KUKA KRL program: MyProgram_294().src

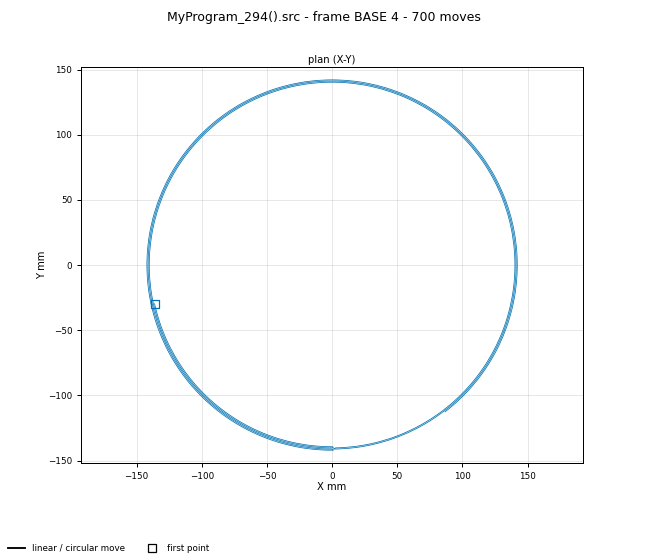
[picture p0: tool path of MyProgram_294().src in frame BASE 4, 700 of 700 moves have a stored position in this frame; points joined in program order, loops and branches not executed]
&ACCESS RVP
&REL 1
&PARAM TEMPLATE = C:\KRC\Roboter\Template\vorgabe
&PARAM EDITMASK = *
DEF MyProgram_294()
; ---- Setting reference (Base) ----
$BASE = BASE_DATA[4]

; --------------------------
; ---- Setting tool (TCP) ----
$TOOL = TOOL_DATA[3]
; --------------------------

$VEL.CP = VEL_APROX_PRINT
Startdeposition()
$VEL.CP = VEL_PRINT
LIN {X -136.1886,Y -29.6785,Z 177,A -164.7897,B 6.5614,C 0.2921,E1 6.4117,E2 257.0139} C_DIS
LIN {X -135.5022,Y -32.6682,Z 177,A -163.4829,B 6.5613,C 0.295,E1 6.4125,E2 255.702} C_DIS
LIN {X -134.5919,Y -36.238,Z 177,A -161.9756,B 6.5611,C 0.2993,E1 6.4136,E2 254.1966} C_DIS
LIN {X -133.5688,Y -39.8487,Z 177,A -160.401,B 6.5609,C 0.3031,E1 6.4148,E2 252.619} C_DIS
LIN {X -132.4479,Y -43.4282,Z 177,A -158.721,B 6.5608,C 0.3057,E1 6.4163,E2 250.9221} C_DIS
LIN {X -130.5858,Y -48.7382,Z 177,A -156.3622,B 6.5605,C 0.3113,E1 6.4185,E2 248.5587} C_DIS
LIN {X -129.1386,Y -52.4536,Z 177,A -154.7567,B 6.5603,C 0.316,E1 6.4201,E2 246.9586} C_DIS
LIN {X -127.4559,Y -56.4207,Z 177,A -152.7896,B 6.5602,C 0.3183,E1 6.4224,E2 244.9671} C_DIS
LIN {X -125.5768,Y -60.4868,Z 177,A -151.0792,B 6.5599,C 0.3246,E1 6.4244,E2 243.2747} C_DIS
LIN {X -123.9871,Y -63.6824,Z 177,A -149.5853,B 6.5597,C 0.3279,E1 6.4263,E2 241.7781} C_DIS
LIN {X -120.2753,Y -70.4446,Z 177,A -146.6108,B 6.5592,C 0.3381,E1 6.4303,E2 238.8308} C_DIS
LIN {X -117.7123,Y -74.649,Z 177,A -144.0898,B 6.5592,C 0.3369,E1 6.4341,E2 236.2462} C_DIS
LIN {X -114.5903,Y -79.3582,Z 177,A -141.8024,B 6.559,C 0.3427,E1 6.4376,E2 233.9644} C_DIS
LIN {X -111.921,Y -83.0801,Z 177,A -139.9675,B 6.5587,C 0.3476,E1 6.4406,E2 232.1365} C_DIS
LIN {X -109.4462,Y -86.3143,Z 177,A -138.2223,B 6.5586,C 0.3504,E1 6.4436,E2 230.3825} C_DIS
LIN {X -106.5575,Y -89.8563,Z 177,A -136.3073,B 6.5584,C 0.3539,E1 6.4471,E2 228.4635} C_DIS
LIN {X -103.5566,Y -93.2993,Z 177,A -134.3994,B 6.5582,C 0.3575,E1 6.4506,E2 226.5522} C_DIS
LIN {X -100.555,Y -96.5264,Z 177,A -132.5532,B 6.558,C 0.3607,E1 6.4541,E2 224.7019} C_DIS
LIN {X -97.3293,Y -99.7782,Z 177,A -130.6364,B 6.5578,C 0.3639,E1 6.458,E2 222.7812} C_DIS
LIN {X -93.9858,Y -102.9341,Z 177,A -128.6876,B 6.5577,C 0.3667,E1 6.462,E2 220.8251} C_DIS
LIN {X -90.5246,Y -105.9904,Z 177,A -126.7715,B 6.5575,C 0.3698,E1 6.466,E2 218.9069} C_DIS
LIN {X -86.9356,Y -108.9531,Z 177,A -124.8461,B 6.5573,C 0.373,E1 6.4702,E2 216.9803} C_DIS
LIN {X -83.3113,Y -111.7488,Z 177,A -122.5359,B 6.5575,C 0.3704,E1 6.4755,E2 214.6138} C_DIS
LIN {X -79.6539,Y -114.3842,Z 177,A -121.0582,B 6.557,C 0.3783,E1 6.4787,E2 213.1858} C_DIS
LIN {X -76.0946,Y -116.7827,Z 177,A -119.334,B 6.5568,C 0.3814,E1 6.4827,E2 211.4669} C_DIS
LIN {X -73.4203,Y -118.4824,Z 177,A -117.9768,B 6.5568,C 0.3825,E1 6.486,E2 210.1027} C_DIS
LIN {X -69.5459,Y -120.7975,Z 177,A -116.113,B 6.5566,C 0.3849,E1 6.4905,E2 208.2377} C_DIS
LIN {X -65.5857,Y -122.9929,Z 177,A -114.0349,B 6.5566,C 0.3843,E1 6.4956,E2 206.131} C_DIS
LIN {X -60.1602,Y -125.7329,Z 177,A -112.0219,B 6.5561,C 0.3939,E1 6.5005,E2 204.1818} C_DIS
LIN {X -56.9114,Y -127.2364,Z 177,A -110.2509,B 6.5562,C 0.3914,E1 6.5051,E2 202.3712} C_DIS
LIN {X -53.2044,Y -128.8317,Z 177,A -108.6402,B 6.5562,C 0.3937,E1 6.5093,E2 200.7667} C_DIS
LIN {X -49.6793,Y -130.2332,Z 177,A -106.9373,B 6.5562,C 0.3932,E1 6.5137,E2 199.0448} C_DIS
LIN {X -46.3018,Y -131.4711,Z 177,A -105.6473,B 6.5559,C 0.3971,E1 6.5171,E2 197.7795} C_DIS
LIN {X -43.7304,Y -132.3472,Z 177,A -104.4709,B 6.5559,C 0.3971,E1 6.5202,E2 196.5949} C_DIS
LIN {X -40.4619,Y -133.3829,Z 177,A -103.0141,B 6.5559,C 0.3975,E1 6.5241,E2 195.1316} C_DIS
LIN {X -34.6228,Y -135.0164,Z 177,A -100.724,B 6.5556,C 0.402,E1 6.5302,E2 192.8676} C_DIS
LIN {X -30.5072,Y -136.0062,Z 177,A -98.6594,B 6.5558,C 0.3982,E1 6.5359,E2 190.7597} C_DIS
LIN {X -26.4921,Y -136.8443,Z 177,A -96.9236,B 6.5558,C 0.3982,E1 6.5407,E2 189.0168} C_DIS
LIN {X -21.8811,Y -137.6576,Z 177,A -95.2757,B 6.5555,C 0.403,E1 6.5451,E2 187.405} C_DIS
LIN {X -19.1338,Y -138.0665,Z 177,A -93.9305,B 6.5557,C 0.4003,E1 6.5489,E2 186.0325} C_DIS
LIN {X -15.0645,Y -138.5684,Z 177,A -92.3262,B 6.5557,C 0.4019,E1 6.5534,E2 184.4383} C_DIS
LIN {X -11.5684,Y -138.904,Z 177,A -90.8501,B 6.5557,C 0.4016,E1 6.5575,E2 182.9572} C_DIS
LIN {X -7.1704,Y -139.2004,Z 177,A -89.0559,B 6.5557,C 0.402,E1 6.5625,E2 181.1646} C_DIS
LIN {X -3.2385,Y -139.3487,Z 177,A -87.4999,B 6.5556,C 0.4028,E1 6.5668,E2 179.6161} C_DIS
LIN {X 0.4018,Y -139.3849,Z 177,A -85.9175,B 6.5556,C 0.4014,E1 6.5713,E2 178.0216} C_DIS
LIN {X 0.4018,Y -139.3849,Z 177,A -85.9175,B 6.5556,C 0.4014,E1 6.5713,E2 178.0216} C_DIS
Enddeposition()
LIN {X 1.0085,Y -140.2847,Z 177,A -86.2982,B 6.5725,C 0.4147,E1 6.5876,E2 178.5133} C_DIS
Startdeposition()
$VEL.CP = VEL_PRINT
LIN {X -2.8125,Y -140.2623,Z 177,A -87.858,B 6.5725,C 0.4149,E1 6.5832,E2 180.0737} C_DIS
LIN {X -6.743,Y -140.1278,Z 177,A -89.5284,B 6.5725,C 0.4159,E1 6.5785,E2 181.7533} C_DIS
LIN {X -10.175,Y -139.9201,Z 177,A -90.9101,B 6.5725,C 0.4154,E1 6.5747,E2 183.1326} C_DIS
LIN {X -14.267,Y -139.5642,Z 177,A -92.617,B 6.5725,C 0.4156,E1 6.5699,E2 184.8441} C_DIS
LIN {X -18.2788,Y -139.0936,Z 177,A -94.2448,B 6.5725,C 0.4149,E1 6.5654,E2 186.4696} C_DIS
LIN {X -22.4184,Y -138.4883,Z 177,A -96.1778,B 6.5723,C 0.4176,E1 6.56,E2 188.4327} C_DIS
LIN {X -27.1842,Y -137.6328,Z 177,A -97.9321,B 6.5726,C 0.4136,E1 6.5553,E2 190.1582} C_DIS
LIN {X -29.7523,Y -137.0983,Z 177,A -99.4764,B 6.5722,C 0.4199,E1 6.5509,E2 191.7649} C_DIS
LIN {X -34.063,Y -136.092,Z 177,A -101.4743,B 6.5721,C 0.4215,E1 6.5454,E2 193.788} C_DIS
LIN {X -39.2291,Y -134.693,Z 177,A -103.0526,B 6.5727,C 0.4114,E1 6.5414,E2 195.2874} C_DIS
LIN {X -42.7662,Y -133.6119,Z 177,A -104.4674,B 6.5729,C 0.409,E1 6.5376,E2 196.6899} C_DIS
LIN {X -45.7296,Y -132.627,Z 177,A -105.8806,B 6.5729,C 0.4099,E1 6.5338,E2 198.1214} C_DIS
LIN {X -50.0559,Y -131.0578,Z 177,A -107.8843,B 6.5729,C 0.4099,E1 6.5285,E2 200.1417} C_DIS
LIN {X -53.8578,Y -129.5394,Z 177,A -109.371,B 6.5731,C 0.4057,E1 6.5248,E2 201.6042} C_DIS
LIN {X -57.9887,Y -127.7457,Z 177,A -111.3634,B 6.5731,C 0.4059,E1 6.5196,E2 203.617} C_DIS
LIN {X -61.8692,Y -125.9098,Z 177,A -113.4842,B 6.5729,C 0.4089,E1 6.5142,E2 205.7859} C_DIS
LIN {X -65.798,Y -123.9035,Z 177,A -114.8633,B 6.5734,C 0.401,E1 6.5109,E2 207.1099} C_DIS
LIN {X -69.5973,Y -121.8106,Z 177,A -116.6692,B 6.5734,C 0.3991,E1 6.5065,E2 208.9203} C_DIS
LIN {X -73.3729,Y -119.5744,Z 177,A -118.3934,B 6.5737,C 0.3958,E1 6.5024,E2 210.6356} C_DIS
LIN {X -76.9211,Y -117.3236,Z 177,A -120.2857,B 6.5737,C 0.3956,E1 6.4979,E2 212.5509} C_DIS
LIN {X -79.8082,Y -115.3794,Z 177,A -122.1332,B 6.5735,C 0.3991,E1 6.4935,E2 214.4538} C_DIS
LIN {X -83.5517,Y -112.6978,Z 177,A -123.6266,B 6.574,C 0.391,E1 6.4903,E2 215.8966} C_DIS
LIN {X -87.2512,Y -109.8583,Z 177,A -125.5322,B 6.5742,C 0.3878,E1 6.4861,E2 217.802} C_DIS
LIN {X -90.6845,Y -107.042,Z 177,A -127.391,B 6.5743,C 0.3852,E1 6.4821,E2 219.6664} C_DIS
LIN {X -94.1044,Y -104.0482,Z 177,A -129.264,B 6.5745,C 0.382,E1 6.4782,E2 221.5413} C_DIS
LIN {X -97.3565,Y -101.012,Z 177,A -131.1315,B 6.5747,C 0.3792,E1 6.4744,E2 223.4149} C_DIS
LIN {X -100.5963,Y -97.7858,Z 177,A -132.9829,B 6.5749,C 0.3753,E1 6.4707,E2 225.2637} C_DIS
LIN {X -103.5666,Y -94.6348,Z 177,A -134.8172,B 6.575,C 0.3726,E1 6.4672,E2 227.1061} C_DIS
LIN {X -106.631,Y -91.1679,Z 177,A -136.7244,B 6.5752,C 0.3688,E1 6.4637,E2 229.0149} C_DIS
LIN {X -109.532,Y -87.6612,Z 177,A -138.6414,B 6.5754,C 0.3655,E1 6.4603,E2 230.9388} C_DIS
LIN {X -112.3124,Y -84.0694,Z 177,A -140.5108,B 6.5756,C 0.3616,E1 6.4572,E2 232.8094} C_DIS
LIN {X -114.9528,Y -80.4213,Z 177,A -142.3794,B 6.5759,C 0.3578,E1 6.4541,E2 234.681} C_DIS
LIN {X -117.1431,Y -77.1953,Z 177,A -144.0543,B 6.5759,C 0.3551,E1 6.4515,E2 236.3659} C_DIS
LIN {X -119.6121,Y -73.3114,Z 177,A -145.7907,B 6.5763,C 0.3488,E1 6.449,E2 238.0829} C_DIS
LIN {X -123.8959,Y -65.8125,Z 177,A -149.4945,B 6.5767,C 0.3424,E1 6.4439,E2 241.808} C_DIS
LIN {X -125.6351,Y -62.4261,Z 177,A -151.0129,B 6.5769,C 0.338,E1 6.442,E2 243.3209} C_DIS
LIN {X -127.1911,Y -59.1911,Z 177,A -152.4543,B 6.5771,C 0.334,E1 6.4403,E2 244.7583} C_DIS
LIN {X -128.6405,Y -55.9712,Z 177,A -153.9384,B 6.5773,C 0.3307,E1 6.4386,E2 246.2469} C_DIS
LIN {X -130.8187,Y -50.671,Z 177,A -156.8492,B 6.5773,C 0.3313,E1 6.4355,E2 249.2297} C_DIS
LIN {X -132.3843,Y -46.4297,Z 177,A -158.2114,B 6.5778,C 0.3207,E1 6.4343,E2 250.5287} C_DIS
LIN {X -133.6222,Y -42.7338,Z 177,A -159.731,B 6.578,C 0.3155,E1 6.433,E2 252.0379} C_DIS
LIN {X -134.5625,Y -39.6748,Z 177,A -161.1596,B 6.5781,C 0.3134,E1 6.4318,E2 253.4813} C_DIS
LIN {X -135.53,Y -36.2316,Z 177,A -162.6621,B 6.5783,C 0.3099,E1 6.4307,E2 254.9882} C_DIS
LIN {X -136.2845,Y -33.2837,Z 177,A -163.8535,B 6.5785,C 0.3059,E1 6.4299,E2 256.1722} C_DIS
LIN {X -137.0587,Y -29.9357,Z 177,A -165.4547,B 6.5785,C 0.3043,E1 6.4289,E2 257.7977} C_DIS
LIN {X -137.8097,Y -26.2605,Z 177,A -167.033,B 6.5787,C 0.3005,E1 6.428,E2 259.3809} C_DIS
LIN {X -138.6022,Y -21.6941,Z 177,A -168.7747,B 6.579,C 0.2935,E1 6.4272,E2 261.1019} C_DIS
LIN {X -139.1207,Y -18.0721,Z 177,A -170.3783,B 6.5792,C 0.2905,E1 6.4266,E2 262.7184} C_DIS
LIN {X -139.8977,Y -10.4823,Z 177,A -173.7243,B 6.5794,C 0.2843,E1 6.4257,E2 266.0915} C_DIS
LIN {X -140.2454,Y -3.5444,Z 177,A -177.3186,B 6.5794,C 0.2848,E1 6.4254,E2 269.7794} C_DIS
LIN {X -140.2664,Y 2.5688,Z 177,A -178.7161,B 6.5802,C 0.2651,E1 6.4254,E2 271.0353} C_DIS
LIN {X -139.9234,Y 10.1302,Z 177,A 178.0725,B 6.5805,C 0.2577,E1 6.4258,E2 274.2598} C_DIS
LIN {X -139.2431,Y 17.1104,Z 177,A 174.739,B 6.5806,C 0.255,E1 6.4268,E2 277.6509} C_DIS
LIN {X -138.3679,Y 23.1403,Z 177,A 171.8862,B 6.5807,C 0.252,E1 6.428,E2 280.5476} C_DIS
LIN {X -137.6263,Y 27.216,Z 177,A 170.4757,B 6.581,C 0.2441,E1 6.4287,E2 281.9211} C_DIS
LIN {X -136.9099,Y 30.6138,Z 177,A 169.0511,B 6.5812,C 0.2402,E1 6.4296,E2 283.3452} C_DIS
LIN {X -136.0591,Y 34.1924,Z 177,A 167.6831,B 6.5814,C 0.2344,E1 6.4305,E2 284.6948} C_DIS
LIN {X -135.1271,Y 37.7063,Z 177,A 166.2172,B 6.5815,C 0.2301,E1 6.4315,E2 286.157} C_DIS
LIN {X -134.2419,Y 40.7467,Z 177,A 164.7417,B 6.5815,C 0.2286,E1 6.4327,E2 287.6544} C_DIS
LIN {X -133.1815,Y 44.0888,Z 177,A 163.3748,B 6.5817,C 0.2239,E1 6.4339,E2 289.0117} C_DIS
LIN {X -131.9466,Y 47.6568,Z 177,A 161.6628,B 6.5818,C 0.2217,E1 6.4355,E2 290.7439} C_DIS
LIN {X -130.9111,Y 50.4334,Z 177,A 160.116,B 6.5818,C 0.2224,E1 6.4371,E2 292.3319} C_DIS
LIN {X -129.5508,Y 53.8303,Z 177,A 158.8562,B 6.582,C 0.2157,E1 6.4384,E2 293.5609} C_DIS
LIN {X -128.054,Y 57.2994,Z 177,A 157.0507,B 6.582,C 0.2147,E1 6.4405,E2 295.3979} C_DIS
LIN {X -126.5856,Y 60.4743,Z 177,A 156.2293,B 6.5824,C 0.2039,E1 6.4413,E2 296.1414} C_DIS
LIN {X -123.4294,Y 66.6851,Z 177,A 152.923,B 6.5824,C 0.2021,E1 6.4456,E2 299.5036} C_DIS
LIN {X -121.1896,Y 70.6744,Z 177,A 151.0247,B 6.5826,C 0.1977,E1 6.4483,E2 301.4039} C_DIS
LIN {X -118.9135,Y 74.4401,Z 177,A 149.1789,B 6.5826,C 0.1939,E1 6.451,E2 303.2542} C_DIS
LIN {X -116.4482,Y 78.2406,Z 177,A 147.2803,B 6.5828,C 0.1901,E1 6.4539,E2 305.1572} C_DIS
LIN {X -113.8534,Y 81.9707,Z 177,A 145.3894,B 6.5829,C 0.1861,E1 6.4569,E2 307.0508} C_DIS
LIN {X -111.5269,Y 85.1079,Z 177,A 143.6904,B 6.5829,C 0.1837,E1 6.4598,E2 308.7614} C_DIS
LIN {X -108.3748,Y 89.088,Z 177,A 141.8945,B 6.5832,C 0.1757,E1 6.4629,E2 310.5205} C_DIS
LIN {X -104.715,Y 93.362,Z 177,A 138.5732,B 6.583,C 0.1831,E1 6.4693,E2 313.9674} C_DIS
LIN {X -100.3605,Y 98.0278,Z 177,A 136.9969,B 6.5835,C 0.1652,E1 6.4721,E2 315.4129} C_DIS
LIN {X -97.366,Y 101.0014,Z 177,A 134.8187,B 6.5835,C 0.1673,E1 6.4765,E2 317.6467} C_DIS
LIN {X -90.5016,Y 107.1973,Z 177,A 131.1066,B 6.5836,C 0.1594,E1 6.4842,E2 321.3474} C_DIS
LIN {X -85.6784,Y 111.0897,Z 177,A 128.1756,B 6.5836,C 0.1598,E1 6.4908,E2 324.3261} C_DIS
LIN {X -82.3284,Y 113.5942,Z 177,A 126.7409,B 6.5838,C 0.1535,E1 6.4939,E2 325.7253} C_DIS
LIN {X -78.3518,Y 116.3732,Z 177,A 124.7895,B 6.5838,C 0.15,E1 6.4984,E2 327.6714} C_DIS
LIN {X -74.5441,Y 118.8484,Z 177,A 122.9372,B 6.5839,C 0.1471,E1 6.5027,E2 329.5219} C_DIS
LIN {X -70.8056,Y 121.1126,Z 177,A 121.1103,B 6.5839,C 0.145,E1 6.5071,E2 331.3525} C_DIS
LIN {X -67.0507,Y 123.2308,Z 177,A 119.354,B 6.584,C 0.1425,E1 6.5114,E2 333.107} C_DIS
LIN {X -63.9541,Y 124.864,Z 177,A 118.0702,B 6.584,C 0.1387,E1 6.5146,E2 334.3712} C_DIS
LIN {X -59.7043,Y 126.9534,Z 177,A 115.932,B 6.584,C 0.139,E1 6.52,E2 336.5336} C_DIS
LIN {X -56.2081,Y 128.5381,Z 177,A 114.5409,B 6.5842,C 0.1349,E1 6.5235,E2 337.9015} C_DIS
LIN {X -54.0951,Y 129.4402,Z 177,A 113.0331,B 6.584,C 0.1413,E1 6.5276,E2 339.4795} C_DIS
LIN {X -49.957,Y 131.0954,Z 177,A 111.6943,B 6.5842,C 0.1331,E1 6.5309,E2 340.7572} C_DIS
LIN {X -46.3635,Y 132.4073,Z 177,A 110.118,B 6.5842,C 0.1318,E1 6.535,E2 342.3341} C_DIS
LIN {X -42.7693,Y 133.6109,Z 177,A 108.5781,B 6.5842,C 0.1303,E1 6.5391,E2 343.8719} C_DIS
LIN {X -40.1654,Y 134.4189,Z 177,A 107.3146,B 6.5842,C 0.1315,E1 6.5425,E2 345.1535} C_DIS
LIN {X -35.8988,Y 135.6187,Z 177,A 105.4528,B 6.5842,C 0.1308,E1 6.5476,E2 347.0206} C_DIS
LIN {X -31.5,Y 136.7075,Z 177,A 103.751,B 6.5843,C 0.1276,E1 6.5521,E2 348.7026} C_DIS
LIN {X -26.0009,Y 137.8594,Z 177,A 101.4275,B 6.5843,C 0.1267,E1 6.5585,E2 351.0283} C_DIS
LIN {X -19.8062,Y 138.8844,Z 177,A 98.8473,B 6.5843,C 0.1258,E1 6.5656,E2 353.6091} C_DIS
LIN {X -16.1577,Y 139.3567,Z 177,A 97.3523,B 6.5843,C 0.1252,E1 6.5698,E2 355.1024} C_DIS
LIN {X -10.6382,Y 139.8863,Z 177,A 95.0449,B 6.5843,C 0.1252,E1 6.5762,E2 357.414} C_DIS
LIN {X -6.0192,Y 140.1616,Z 177,A 93.1305,B 6.5843,C 0.1254,E1 6.5815,E2 359.3306} C_DIS
LIN {X -2.6617,Y 140.2649,Z 177,A 91.7806,B 6.5843,C 0.125,E1 6.5853,E2 360.677} C_DIS
LIN {X 1.2875,Y 140.2848,Z 177,A 90.1404,B 6.5843,C 0.1254,E1 6.5899,E2 362.32} C_DIS
LIN {X 5.4175,Y 140.1851,Z 177,A 88.5025,B 6.5843,C 0.1249,E1 6.5944,E2 363.951} C_DIS
LIN {X 9.1341,Y 139.9929,Z 177,A 86.9392,B 6.5843,C 0.1258,E1 6.5988,E2 365.5191} C_DIS
LIN {X 13.3698,Y 139.6511,Z 177,A 85.2082,B 6.5843,C 0.1262,E1 6.6036,E2 367.2489} C_DIS
LIN {X 16.9885,Y 139.2576,Z 177,A 83.1093,B 6.5841,C 0.1357,E1 6.6097,E2 369.4234} C_DIS
LIN {X 22.4493,Y 138.4829,Z 177,A 81.6183,B 6.5843,C 0.1255,E1 6.6135,E2 370.8189} C_DIS
LIN {X 26.1488,Y 137.8311,Z 177,A 80.2557,B 6.5843,C 0.1237,E1 6.6172,E2 372.1595} C_DIS
LIN {X 29.9376,Y 137.0583,Z 177,A 78.3564,B 6.5843,C 0.1295,E1 6.6225,E2 374.0986} C_DIS
LIN {X 36.1305,Y 135.5569,Z 177,A 75.9146,B 6.5843,C 0.1289,E1 6.6291,E2 376.5197} C_DIS
LIN {X 39.0885,Y 134.7342,Z 177,A 74.5832,B 6.5843,C 0.131,E1 6.6327,E2 377.8606} C_DIS
LIN {X 42.8233,Y 133.5936,Z 177,A 73.0978,B 6.5843,C 0.1307,E1 6.6366,E2 379.3319} C_DIS
LIN {X 45.4483,Y 132.7246,Z 177,A 71.8929,B 6.5842,C 0.133,E1 6.6398,E2 380.5461} C_DIS
LIN {X 49.166,Y 131.3917,Z 177,A 70.3302,B 6.5842,C 0.1338,E1 6.6439,E2 382.1022} C_DIS
LIN {X 52.1938,Y 130.2188,Z 177,A 68.9022,B 6.5842,C 0.1368,E1 6.6476,E2 383.5429} C_DIS
LIN {X 55.0349,Y 129.0453,Z 177,A 67.6015,B 6.5841,C 0.1389,E1 6.651,E2 384.8492} C_DIS
LIN {X 58.7087,Y 127.4141,Z 177,A 66.2366,B 6.5841,C 0.1365,E1 6.6544,E2 386.1792} C_DIS
LIN {X 62.8623,Y 125.4197,Z 177,A 64.0354,B 6.584,C 0.1439,E1 6.66,E2 388.4205} C_DIS
LIN {X 67.0569,Y 123.2274,Z 177,A 62.257,B 6.584,C 0.1441,E1 6.6643,E2 390.1795} C_DIS
LIN {X 70.8277,Y 121.0996,Z 177,A 60.4983,B 6.584,C 0.1465,E1 6.6686,E2 391.937} C_DIS
LIN {X 74.6827,Y 118.7609,Z 177,A 58.6728,B 6.5839,C 0.149,E1 6.6729,E2 393.7606} C_DIS
LIN {X 77.762,Y 116.7677,Z 177,A 56.9406,B 6.5837,C 0.1552,E1 6.677,E2 395.5223} C_DIS
LIN {X 80.7904,Y 114.6931,Z 177,A 55.7179,B 6.5837,C 0.1531,E1 6.6797,E2 396.7104} C_DIS
LIN {X 84.4748,Y 112.0072,Z 177,A 53.886,B 6.5837,C 0.1558,E1 6.6838,E2 398.5388} C_DIS
LIN {X 88.1049,Y 109.1748,Z 177,A 52.0707,B 6.5837,C 0.1581,E1 6.6878,E2 400.346} C_DIS
LIN {X 91.384,Y 106.4454,Z 177,A 50.291,B 6.5836,C 0.1619,E1 6.6916,E2 402.1308} C_DIS
LIN {X 93.6819,Y 104.4285,Z 177,A 48.8027,B 6.5834,C 0.1683,E1 6.6948,E2 403.6496} C_DIS
LIN {X 96.4608,Y 101.8673,Z 177,A 47.3522,B 6.5834,C 0.1698,E1 6.6977,E2 405.0887} C_DIS
LIN {X 98.8762,Y 99.5243,Z 177,A 46.2222,B 6.5834,C 0.1685,E1 6.6999,E2 406.1882} C_DIS
LIN {X 101.9908,Y 96.3301,Z 177,A 44.4306,B 6.5834,C 0.1717,E1 6.7033,E2 407.9765} C_DIS
LIN {X 104.8849,Y 93.1712,Z 177,A 42.6508,B 6.5832,C 0.1759,E1 6.7067,E2 409.7606} C_DIS
LIN {X 107.5781,Y 90.0476,Z 177,A 40.7504,B 6.583,C 0.1833,E1 6.7101,E2 411.6889} C_DIS
LIN {X 110.006,Y 87.0656,Z 177,A 39.293,B 6.583,C 0.1849,E1 6.7126,E2 413.1326} C_DIS
LIN {X 112.0134,Y 84.4666,Z 177,A 38.1872,B 6.583,C 0.1839,E1 6.7145,E2 414.2091} C_DIS
LIN {X 114.6729,Y 80.8192,Z 177,A 36.3902,B 6.5829,C 0.1874,E1 6.7174,E2 416.0009} C_DIS
LIN {X 117.0596,Y 77.3221,Z 177,A 34.6716,B 6.5828,C 0.1913,E1 6.7201,E2 417.7188} C_DIS
LIN {X 119.402,Y 73.6538,Z 177,A 32.9779,B 6.5827,C 0.1942,E1 6.7226,E2 419.4027} C_DIS
LIN {X 122.8059,Y 67.8259,Z 177,A 30.2512,B 6.5825,C 0.2005,E1 6.7264,E2 422.127} C_DIS
LIN {X 124.8498,Y 63.982,Z 177,A 28.6087,B 6.5825,C 0.2026,E1 6.7285,E2 423.753} C_DIS
LIN {X 126.5611,Y 60.5255,Z 177,A 26.8637,B 6.5822,C 0.2096,E1 6.7306,E2 425.5205} C_DIS
LIN {X 128.5353,Y 56.2145,Z 177,A 25.1986,B 6.5822,C 0.2099,E1 6.7325,E2 427.152} C_DIS
LIN {X 129.4318,Y 54.1153,Z 177,A 23.6668,B 6.5818,C 0.2229,E1 6.7342,E2 428.7608} C_DIS
LIN {X 131.2034,Y 49.6687,Z 177,A 22.2834,B 6.5819,C 0.2181,E1 6.7355,E2 430.0726} C_DIS
LIN {X 132.2869,Y 46.7107,Z 177,A 20.862,B 6.5817,C 0.2239,E1 6.7369,E2 431.5121} C_DIS
LIN {X 133.5959,Y 42.8163,Z 177,A 19.4766,B 6.5817,C 0.2233,E1 6.7381,E2 432.8609} C_DIS
LIN {X 134.501,Y 39.8848,Z 177,A 18.0948,B 6.5816,C 0.229,E1 6.7392,E2 434.2602} C_DIS
LIN {X 135.5067,Y 36.319,Z 177,A 16.6912,B 6.5815,C 0.2312,E1 6.7402,E2 435.6507} C_DIS
LIN {X 136.6249,Y 31.8615,Z 177,A 14.7687,B 6.5813,C 0.2372,E1 6.7415,E2 437.5804} C_DIS
LIN {X 137.538,Y 27.6502,Z 177,A 13.0851,B 6.5812,C 0.2408,E1 6.7425,E2 439.2554} C_DIS
LIN {X 138.3059,Y 23.5119,Z 177,A 11.4808,B 6.581,C 0.2436,E1 6.7433,E2 440.8461} C_DIS
LIN {X 139.4436,Y 15.3878,Z 177,A 8.2508,B 6.5808,C 0.251,E1 6.7445,E2 444.0632} C_DIS
LIN {X 139.7807,Y 11.9399,Z 177,A 6.7331,B 6.5805,C 0.2568,E1 6.7449,E2 445.5952} C_DIS
LIN {X 140.0808,Y 7.6784,Z 177,A 4.9926,B 6.5804,C 0.2618,E1 6.7452,E2 447.3367} C_DIS
LIN {X 140.2349,Y 3.9226,Z 177,A 3.5309,B 6.5802,C 0.2648,E1 6.7453,E2 448.7901} C_DIS
LIN {X 140.2914,Y -0.3591,Z 177,A 1.7307,B 6.58,C 0.2708,E1 6.7453,E2 450.5984} C_DIS
LIN {X 140.23,Y -4.099,Z 177,A 0.2993,B 6.5799,C 0.2734,E1 6.7453,E2 452.0185} C_DIS
LIN {X 140.0334,Y -8.4773,Z 177,A -1.4237,B 6.5797,C 0.2773,E1 6.745,E2 453.7344} C_DIS
LIN {X 139.6878,Y -12.9868,Z 177,A -3.278,B 6.5795,C 0.2828,E1 6.7446,E2 455.5912} C_DIS
LIN {X 139.258,Y -16.9854,Z 177,A -4.8278,B 6.5794,C 0.2858,E1 6.7441,E2 457.1304} C_DIS
LIN {X 138.708,Y -21.0103,Z 177,A -6.4678,B 6.5792,C 0.2902,E1 6.7434,E2 458.7694} C_DIS
LIN {X 138.0213,Y -25.1285,Z 177,A -8.6193,B 6.5786,C 0.303,E1 6.7423,E2 460.9802} C_DIS
LIN {X 137.1268,Y -29.6204,Z 177,A -9.7664,B 6.5789,C 0.2953,E1 6.7418,E2 462.0351} C_DIS
LIN {X 136.5856,Y -32.0302,Z 177,A -11.3913,B 6.5783,C 0.3092,E1 6.7407,E2 463.741} C_DIS
LIN {X 135.5504,Y -36.1551,Z 177,A -13.0081,B 6.5782,C 0.3119,E1 6.7395,E2 465.3438} C_DIS
LIN {X 134.4743,Y -39.9762,Z 177,A -14.3777,B 6.5782,C 0.3119,E1 6.7385,E2 466.6824} C_DIS
LIN {X 133.1782,Y -44.0987,Z 177,A -15.9265,B 6.5782,C 0.3129,E1 6.7371,E2 468.2046} C_DIS
LIN {X 132.0542,Y -47.3583,Z 177,A -17.3572,B 6.5779,C 0.3171,E1 6.7358,E2 469.6395} C_DIS
LIN {X 130.4517,Y -51.6151,Z 177,A -19.241,B 6.5777,C 0.3226,E1 6.7339,E2 471.5286} C_DIS
LIN {X 128.863,Y -55.4566,Z 177,A -20.7476,B 6.5777,C 0.3237,E1 6.7323,E2 473.0117} C_DIS
LIN {X 127.4057,Y -58.7271,Z 177,A -22.2062,B 6.5774,C 0.3275,E1 6.7306,E2 474.4712} C_DIS
LIN {X 126.0083,Y -61.6696,Z 177,A -23.7783,B 6.577,C 0.3353,E1 6.7287,E2 476.0762} C_DIS
LIN {X 123.3932,Y -66.7525,Z 177,A -25.8984,B 6.577,C 0.3375,E1 6.726,E2 478.1705} C_DIS
LIN {X 121.2012,Y -70.6544,Z 177,A -27.7318,B 6.5767,C 0.3423,E1 6.7234,E2 480.0063} C_DIS
LIN {X 118.2134,Y -75.5458,Z 177,A -30.0534,B 6.5764,C 0.3477,E1 6.72,E2 482.3276} C_DIS
LIN {X 115.9741,Y -78.9413,Z 177,A -32.0552,B 6.5759,C 0.3577,E1 6.7168,E2 484.3755} C_DIS
LIN {X 113.3323,Y -82.6897,Z 177,A -33.4777,B 6.576,C 0.3543,E1 6.7146,E2 485.741} C_DIS
LIN {X 109.3545,Y -87.882,Z 177,A -36.0745,B 6.5758,C 0.3592,E1 6.7101,E2 488.3305} C_DIS
LIN {X 106.6221,Y -91.1784,Z 177,A -37.7708,B 6.5756,C 0.3622,E1 6.7071,E2 490.0215} C_DIS
LIN {X 102.7203,Y -95.5518,Z 177,A -40.3226,B 6.5752,C 0.3702,E1 6.7022,E2 492.5963} C_DIS
LIN {X 99.269,Y -99.1332,Z 177,A -42.153,B 6.5752,C 0.371,E1 6.6987,E2 494.4022} C_DIS
LIN {X 96.2538,Y -102.0628,Z 177,A -43.8498,B 6.5749,C 0.3742,E1 6.6953,E2 496.0979} C_DIS
LIN {X 92.7058,Y -105.2963,Z 177,A -45.9615,B 6.5746,C 0.3807,E1 6.6908,E2 498.2313} C_DIS
LIN {X 88.5945,Y -108.7781,Z 177,A -47.9877,B 6.5745,C 0.3819,E1 6.6865,E2 500.2365} C_DIS
LIN {X 85.2146,Y -111.4454,Z 177,A -49.5724,B 6.5745,C 0.3822,E1 6.6831,E2 501.7999} C_DIS
LIN {X 82.018,Y -113.8189,Z 177,A -51.858,B 6.5737,C 0.3963,E1 6.6777,E2 504.1734} C_DIS
LIN {X 77.6187,Y -116.8634,Z 177,A -53.2103,B 6.5743,C 0.3859,E1 6.6749,E2 505.4182} C_DIS
LIN {X 72.6109,Y -120.0386,Z 177,A -56.084,B 6.5736,C 0.3974,E1 6.6679,E2 508.3536} C_DIS
LIN {X 69.5653,Y -121.8289,Z 177,A -57.3926,B 6.5736,C 0.3974,E1 6.6648,E2 509.6458} C_DIS
LIN {X 65.3318,Y -124.1483,Z 177,A -59.1044,B 6.5736,C 0.3959,E1 6.6606,E2 511.3248} C_DIS
LIN {X 62.3779,Y -125.6589,Z 177,A -60.4801,B 6.5736,C 0.3982,E1 6.6572,E2 512.7044} C_DIS
LIN {X 59.2232,Y -127.1762,Z 177,A -61.9318,B 6.5734,C 0.4004,E1 6.6535,E2 514.1601} C_DIS
LIN {X 56.3905,Y -128.4592,Z 177,A -63.2881,B 6.5732,C 0.4035,E1 6.65,E2 515.5289} C_DIS
LIN {X 53.2759,Y -129.7823,Z 177,A -64.6574,B 6.5732,C 0.4049,E1 6.6465,E2 516.8975} C_DIS
LIN {X 50.0317,Y -131.0672,Z 177,A -66.0478,B 6.5731,C 0.406,E1 6.6429,E2 518.2845} C_DIS
LIN {X 46.3393,Y -132.4157,Z 177,A -67.4652,B 6.5731,C 0.4047,E1 6.6392,E2 519.6781} C_DIS
LIN {X 42.931,Y -133.5593,Z 177,A -68.9131,B 6.5731,C 0.4058,E1 6.6354,E2 521.1243} C_DIS
LIN {X 38.9298,Y -134.7806,Z 177,A -70.8146,B 6.5728,C 0.4105,E1 6.6302,E2 523.0526} C_DIS
LIN {X 35.8756,Y -135.6249,Z 177,A -72.066,B 6.5728,C 0.4109,E1 6.6269,E2 524.2991} C_DIS
LIN {X 29.8384,Y -137.0797,Z 177,A -74.5403,B 6.5727,C 0.4119,E1 6.6201,E2 526.7669} C_DIS
LIN {X 25.9633,Y -137.8665,Z 177,A -76.1016,B 6.5727,C 0.4121,E1 6.6159,E2 528.3221} C_DIS
LIN {X 22.2732,Y -138.5125,Z 177,A -78.1304,B 6.5721,C 0.4208,E1 6.6101,E2 530.4176} C_DIS
LIN {X 17.8376,Y -139.1515,Z 177,A -79.519,B 6.5725,C 0.4149,E1 6.6064,E2 531.7491} C_DIS
LIN {X 13.4075,Y -139.6474,Z 177,A -81.2307,B 6.5725,C 0.414,E1 6.6017,E2 533.4474} C_DIS
LIN {X 10.3473,Y -139.9076,Z 177,A -82.5275,B 6.5725,C 0.415,E1 6.5981,E2 534.7505} C_DIS
LIN {X 6.2442,Y -140.1528,Z 177,A -84.3049,B 6.5724,C 0.417,E1 6.5931,E2 536.5419} C_DIS
LIN {X 2.6932,Y -140.2643,Z 177,A -85.512,B 6.5726,C 0.4136,E1 6.5898,E2 537.7174} C_DIS
LIN {X 2.6932,Y -140.2643,Z 177,A -85.512,B 6.5726,C 0.4136,E1 6.5898,E2 537.7174} C_DIS
Enddeposition()
LIN {X 1.012,Y -141.1907,Z 177,A -86.1424,B 6.5725,C 0.4166,E1 6.588,E2 538.3737} C_DIS
Startdeposition()
$VEL.CP = VEL_PRINT
LIN {X 4.7836,Y -141.1152,Z 177,A -83.9653,B 6.5731,C 0.4063,E1 6.5943,E2 536.1093} C_DIS
LIN {X 9.5309,Y -140.8743,Z 177,A -82.2574,B 6.5729,C 0.4092,E1 6.599,E2 534.4301} C_DIS
LIN {X 12.4111,Y -140.6488,Z 177,A -81.0777,B 6.5729,C 0.4087,E1 6.6023,E2 533.2488} C_DIS
LIN {X 15.2755,Y -140.3657,Z 177,A -79.9309,B 6.5729,C 0.4085,E1 6.6055,E2 532.1042} C_DIS
LIN {X 18.1867,Y -140.0182,Z 177,A -78.5889,B 6.5731,C 0.4055,E1 6.6093,E2 530.7409} C_DIS
LIN {X 22.375,Y -139.4123,Z 177,A -77.0206,B 6.5731,C 0.407,E1 6.6135,E2 529.1918} C_DIS
LIN {X 27.2146,Y -138.5485,Z 177,A -75.029,B 6.5731,C 0.4057,E1 6.619,E2 527.1994} C_DIS
LIN {X 30.5672,Y -137.848,Z 177,A -72.9898,B 6.5738,C 0.3942,E1 6.6248,E2 525.0715} C_DIS
LIN {X 35.6693,Y -136.6163,Z 177,A -71.4047,B 6.5734,C 0.4013,E1 6.6289,E2 523.5588} C_DIS
LIN {X 41.907,Y -134.833,Z 177,A -68.9053,B 6.5734,C 0.4011,E1 6.6356,E2 521.0755} C_DIS
LIN {X 44.8529,Y -133.8807,Z 177,A -67.6181,B 6.5735,C 0.3993,E1 6.639,E2 519.7833} C_DIS
LIN {X 48.6276,Y -132.5584,Z 177,A -66.0326,B 6.5735,C 0.3982,E1 6.6431,E2 518.2017} C_DIS
LIN {X 51.3576,Y -131.5226,Z 177,A -64.8409,B 6.5737,C 0.3967,E1 6.6463,E2 517.0082} C_DIS
LIN {X 55.361,Y -129.89,Z 177,A -63.1642,B 6.5737,C 0.3959,E1 6.6506,E2 515.3406} C_DIS
LIN {X 58.1589,Y -128.6607,Z 177,A -61.893,B 6.5739,C 0.3938,E1 6.6538,E2 514.0643} C_DIS
LIN {X 61.4404,Y -127.1267,Z 177,A -60.4447,B 6.5739,C 0.3922,E1 6.6575,E2 512.6178} C_DIS
LIN {X 64.3741,Y -125.6655,Z 177,A -59.1227,B 6.5741,C 0.3905,E1 6.6608,E2 511.2957} C_DIS
LIN {X 67.334,Y -124.1069,Z 177,A -57.1772,B 6.5748,C 0.3785,E1 6.6657,E2 509.2698} C_DIS
LIN {X 71.7884,Y -121.5846,Z 177,A -55.7083,B 6.5743,C 0.3857,E1 6.6691,E2 507.8815} C_DIS
LIN {X 75.1826,Y -119.5153,Z 177,A -54.0172,B 6.5746,C 0.3818,E1 6.6731,E2 506.1785} C_DIS
LIN {X 79.1082,Y -116.9538,Z 177,A -52.032,B 6.5748,C 0.3772,E1 6.6778,E2 504.1805} C_DIS
LIN {X 82.9335,Y -114.273,Z 177,A -50.2913,B 6.5748,C 0.3765,E1 6.6817,E2 502.459} C_DIS
LIN {X 86.4075,Y -111.6693,Z 177,A -48.5918,B 6.575,C 0.3744,E1 6.6854,E2 500.7664} C_DIS
LIN {X 89.5517,Y -109.1643,Z 177,A -46.9941,B 6.5751,C 0.3719,E1 6.6889,E2 499.1717} C_DIS
LIN {X 92.7612,Y -106.4502,Z 177,A -45.4441,B 6.5751,C 0.3713,E1 6.6921,E2 497.6411} C_DIS
LIN {X 95.3166,Y -104.1688,Z 177,A -43.9397,B 6.5754,C 0.3665,E1 6.6953,E2 496.1201} C_DIS
LIN {X 98.3415,Y -101.3176,Z 177,A -42.2615,B 6.5756,C 0.3632,E1 6.6987,E2 494.4415} C_DIS
LIN {X 101.3355,Y -98.323,Z 177,A -40.5605,B 6.5758,C 0.3599,E1 6.702,E2 492.7413} C_DIS
LIN {X 103.953,Y -95.5513,Z 177,A -39.1962,B 6.5758,C 0.3598,E1 6.7046,E2 491.4001} C_DIS
LIN {X 106.2487,Y -92.9922,Z 177,A -37.6901,B 6.5761,C 0.3547,E1 6.7074,E2 489.8778} C_DIS
LIN {X 108.8186,Y -89.9712,Z 177,A -36.1215,B 6.5762,C 0.3518,E1 6.7102,E2 488.3132} C_DIS
LIN {X 111.7724,Y -86.274,Z 177,A -33.8286,B 6.5768,C 0.3407,E1 6.7142,E2 485.9683} C_DIS
LIN {X 114.3232,Y -82.8643,Z 177,A -32.6005,B 6.5766,C 0.3456,E1 6.7162,E2 484.8058} C_DIS
LIN {X 116.4744,Y -79.8123,Z 177,A -30.9799,B 6.5768,C 0.34,E1 6.7187,E2 483.1696} C_DIS
LIN {X 118.8966,Y -76.157,Z 177,A -28.9751,B 6.5773,C 0.3316,E1 6.7218,E2 481.1329} C_DIS
LIN {X 120.9132,Y -72.9131,Z 177,A -27.7261,B 6.5772,C 0.3332,E1 6.7236,E2 479.9228} C_DIS
LIN {X 123.234,Y -68.9186,Z 177,A -25.8601,B 6.5774,C 0.3286,E1 6.7262,E2 478.0562} C_DIS
LIN {X 125.538,Y -64.6245,Z 177,A -24.1207,B 6.5774,C 0.3278,E1 6.7284,E2 476.3467} C_DIS
LIN {X 126.8311,Y -62.0468,Z 177,A -22.8622,B 6.5777,C 0.3231,E1 6.73,E2 475.0753} C_DIS
LIN {X 128.3338,Y -58.8757,Z 177,A -21.4677,B 6.5779,C 0.3199,E1 6.7316,E2 473.6834} C_DIS
LIN {X 129.7286,Y -55.7344,Z 177,A -20.1761,B 6.5779,C 0.3181,E1 6.733,E2 472.4042} C_DIS
LIN {X 130.8036,Y -53.1633,Z 177,A -19.1384,B 6.578,C 0.3167,E1 6.7341,E2 471.3779} C_DIS
LIN {X 131.83,Y -50.5667,Z 177,A -17.9292,B 6.5782,C 0.3123,E1 6.7354,E2 470.1575} C_DIS
LIN {X 132.9561,Y -47.5244,Z 177,A -16.598,B 6.5784,C 0.3084,E1 6.7366,E2 468.8231} C_DIS
LIN {X 133.9904,Y -44.5234,Z 177,A -15.3324,B 6.5785,C 0.3053,E1 6.7378,E2 467.5592} C_DIS
LIN {X 136.2839,Y -36.9158,Z 177,A -12.3137,B 6.5788,C 0.3002,E1 6.7401,E2 464.5651} C_DIS
LIN {X 137.0802,Y -33.8441,Z 177,A -10.9201,B 6.579,C 0.2946,E1 6.7411,E2 463.1564} C_DIS
LIN {X 137.851,Y -30.5532,Z 177,A -9.6333,B 6.5791,C 0.2923,E1 6.7419,E2 461.8796} C_DIS
LIN {X 138.6982,Y -26.4317,Z 177,A -7.8931,B 6.5794,C 0.2869,E1 6.7428,E2 460.1334} C_DIS
LIN {X 139.3642,Y -22.6664,Z 177,A -6.4416,B 6.5794,C 0.2843,E1 6.7435,E2 458.6938} C_DIS
LIN {X 139.7839,Y -19.9071,Z 177,A -5.25,B 6.5797,C 0.28,E1 6.744,E2 457.4934} C_DIS
LIN {X 140.3059,Y -15.8315,Z 177,A -3.7194,B 6.5797,C 0.2778,E1 6.7445,E2 455.9795} C_DIS
LIN {X 140.5861,Y -13.0981,Z 177,A -2.6264,B 6.5799,C 0.275,E1 6.7448,E2 454.8883} C_DIS
LIN {X 140.8342,Y -10.0814,Z 177,A -1.3377,B 6.5801,C 0.2703,E1 6.7451,E2 453.5907} C_DIS
LIN {X 141.0489,Y -6.4418,Z 177,A 0.0374,B 6.5801,C 0.268,E1 6.7453,E2 452.2282} C_DIS
LIN {X 141.1548,Y -3.391,Z 177,A 1.3731,B 6.5804,C 0.2627,E1 6.7453,E2 450.8786} C_DIS
LIN {X 141.1921,Y 0.9576,Z 177,A 2.9639,B 6.5804,C 0.2608,E1 6.7453,E2 449.3092} C_DIS
LIN {X 141.1376,Y 4.0089,Z 177,A 4.2533,B 6.5806,C 0.2563,E1 6.7453,E2 448.0121} C_DIS
LIN {X 140.9945,Y 7.523,Z 177,A 5.5755,B 6.5807,C 0.2541,E1 6.7451,E2 446.7027} C_DIS
LIN {X 140.7909,Y 10.6747,Z 177,A 6.9941,B 6.5809,C 0.248,E1 6.7448,E2 445.2649} C_DIS
LIN {X 140.4491,Y 14.501,Z 177,A 8.3118,B 6.5809,C 0.248,E1 6.7445,E2 443.9778} C_DIS
LIN {X 139.8196,Y 19.6577,Z 177,A 10.33,B 6.5811,C 0.2436,E1 6.7438,E2 441.9699} C_DIS
LIN {X 139.4441,Y 22.1699,Z 177,A 11.4252,B 6.5813,C 0.2395,E1 6.7433,E2 440.8655} C_DIS
LIN {X 138.8196,Y 25.7965,Z 177,A 12.8808,B 6.5813,C 0.236,E1 6.7426,E2 439.4137} C_DIS
LIN {X 138.3518,Y 28.1882,Z 177,A 13.9833,B 6.5816,C 0.2312,E1 6.742,E2 438.2956} C_DIS
LIN {X 137.5437,Y 31.9022,Z 177,A 15.546,B 6.5817,C 0.2265,E1 6.741,E2 436.7291} C_DIS
LIN {X 136.3623,Y 36.6219,Z 177,A 17.3417,B 6.5817,C 0.2243,E1 6.7398,E2 434.9556} C_DIS
LIN {X 135.3686,Y 40.1416,Z 177,A 18.9316,B 6.582,C 0.2183,E1 6.7385,E2 433.3509} C_DIS
LIN {X 134.1638,Y 44.0027,Z 177,A 20.3521,B 6.582,C 0.2178,E1 6.7373,E2 431.9583} C_DIS
LIN {X 133.1571,Y 46.9629,Z 177,A 21.6415,B 6.5821,C 0.214,E1 6.7362,E2 430.6653} C_DIS
LIN {X 131.96,Y 50.228,Z 177,A 23.2098,B 6.5823,C 0.2074,E1 6.7346,E2 429.0756} C_DIS
LIN {X 130.5255,Y 53.8442,Z 177,A 24.672,B 6.5824,C 0.2053,E1 6.7331,E2 427.6277} C_DIS
LIN {X 128.9961,Y 57.4092,Z 177,A 26.0728,B 6.5824,C 0.2043,E1 6.7315,E2 426.2486} C_DIS
LIN {X 126.6323,Y 62.4499,Z 177,A 28.0341,B 6.5824,C 0.2038,E1 6.7293,E2 424.325} C_DIS
LIN {X 125.6603,Y 64.3842,Z 177,A 29.2325,B 6.5827,C 0.1958,E1 6.7277,E2 423.0845} C_DIS
LIN {X 123.661,Y 68.1494,Z 177,A 31.097,B 6.5829,C 0.1891,E1 6.7252,E2 421.2017} C_DIS
LIN {X 121.902,Y 71.2482,Z 177,A 32.3677,B 6.5829,C 0.1887,E1 6.7234,E2 419.9531} C_DIS
LIN {X 119.8421,Y 74.6603,Z 177,A 33.934,B 6.5829,C 0.1856,E1 6.7211,E2 418.3928} C_DIS
LIN {X 117.7272,Y 77.9534,Z 177,A 35.4987,B 6.5831,C 0.1822,E1 6.7187,E2 416.8304} C_DIS
LIN {X 115.2676,Y 81.5457,Z 177,A 37.3024,B 6.5832,C 0.1774,E1 6.7159,E2 415.0212} C_DIS
LIN {X 112.5105,Y 85.3099,Z 177,A 40.1526,B 6.5837,C 0.1564,E1 6.7109,E2 412.0449} C_DIS
LIN {X 107.5222,Y 91.5165,Z 177,A 42.1698,B 6.5834,C 0.1704,E1 6.7075,E2 410.1855} C_DIS
LIN {X 104.9561,Y 94.449,Z 177,A 43.7227,B 6.5834,C 0.1675,E1 6.7046,E2 408.6359} C_DIS
LIN {X 102.5186,Y 97.0891,Z 177,A 45.3045,B 6.5836,C 0.1624,E1 6.7016,E2 407.0377} C_DIS
LIN {X 99.2825,Y 100.3961,Z 177,A 48.1889,B 6.5841,C 0.1413,E1 6.6956,E2 404.0213} C_DIS
LIN {X 93.3926,Y 105.8968,Z 177,A 50.1583,B 6.5837,C 0.1572,E1 6.6919,E2 402.2208} C_DIS
LIN {X 90.3291,Y 108.5222,Z 177,A 51.8988,B 6.5838,C 0.1525,E1 6.6881,E2 400.4668} C_DIS
LIN {X 87.1999,Y 111.0516,Z 177,A 53.6167,B 6.5839,C 0.1481,E1 6.6843,E2 398.7377} C_DIS
LIN {X 83.415,Y 113.9222,Z 177,A 55.5289,B 6.5839,C 0.1451,E1 6.6801,E2 396.8272} C_DIS
LIN {X 79.4463,Y 116.7249,Z 177,A 57.3156,B 6.584,C 0.1449,E1 6.676,E2 395.0641} C_DIS
LIN {X 76.6576,Y 118.5747,Z 177,A 58.7417,B 6.584,C 0.1416,E1 6.6727,E2 393.6292} C_DIS
LIN {X 73.2937,Y 120.6831,Z 177,A 60.399,B 6.5841,C 0.1384,E1 6.6687,E2 391.9658} C_DIS
LIN {X 69.37,Y 122.9803,Z 177,A 62.2252,B 6.5841,C 0.1361,E1 6.6643,E2 390.142} C_DIS
LIN {X 63.8791,Y 125.9175,Z 177,A 64.3161,B 6.5841,C 0.1398,E1 6.6593,E2 388.107} C_DIS
LIN {X 61.3372,Y 127.176,Z 177,A 65.8315,B 6.5843,C 0.1324,E1 6.6554,E2 386.5452} C_DIS
LIN {X 57.8404,Y 128.8032,Z 177,A 67.385,B 6.5843,C 0.1308,E1 6.6514,E2 384.9932} C_DIS
LIN {X 54.7101,Y 130.1639,Z 177,A 68.557,B 6.5843,C 0.1326,E1 6.6485,E2 383.8486} C_DIS
LIN {X 52.4791,Y 131.0793,Z 177,A 69.6937,B 6.5843,C 0.129,E1 6.6455,E2 382.6917} C_DIS
LIN {X 49.1155,Y 132.3768,Z 177,A 71.0736,B 6.5843,C 0.1288,E1 6.6419,E2 381.3227} C_DIS
LIN {X 46.1722,Y 133.4312,Z 177,A 72.3456,B 6.5843,C 0.1276,E1 6.6385,E2 380.0504} C_DIS
LIN {X 43.2079,Y 134.4206,Z 177,A 73.5835,B 6.5843,C 0.1269,E1 6.6353,E2 378.8167} C_DIS
LIN {X 40.2103,Y 135.3485,Z 177,A 74.7871,B 6.5843,C 0.1269,E1 6.6321,E2 377.6223} C_DIS
LIN {X 37.2485,Y 136.1946,Z 177,A 76.4335,B 6.5845,C 0.1198,E1 6.6275,E2 375.9254} C_DIS
LIN {X 34.0023,Y 137.0409,Z 177,A 77.4838,B 6.5845,C 0.1236,E1 6.6248,E2 374.9153} C_DIS
LIN {X 31.0688,Y 137.7341,Z 177,A 78.7436,B 6.5845,C 0.1222,E1 6.6213,E2 373.6511} C_DIS
LIN {X 27.8029,Y 138.4302,Z 177,A 80.1164,B 6.5845,C 0.1212,E1 6.6176,E2 372.2764} C_DIS
LIN {X 24.1154,Y 139.1217,Z 177,A 81.5548,B 6.5845,C 0.1217,E1 6.6136,E2 370.8492} C_DIS
LIN {X 18.937,Y 139.9199,Z 177,A 83.5971,B 6.5845,C 0.122,E1 6.608,E2 368.8182} C_DIS
LIN {X 16.2733,Y 140.2541,Z 177,A 84.7432,B 6.5845,C 0.1208,E1 6.6048,E2 367.6654} C_DIS
LIN {X 13.5297,Y 140.5447,Z 177,A 85.848,B 6.5845,C 0.1206,E1 6.6018,E2 366.5628} C_DIS
LIN {X 10.3267,Y 140.8163,Z 177,A 87.2379,B 6.5845,C 0.119,E1 6.5979,E2 365.1625} C_DIS
LIN {X 6.0694,Y 141.0651,Z 177,A 89.0436,B 6.5845,C 0.1177,E1 6.5928,E2 363.3478} C_DIS
LIN {X 2.3862,Y 141.1743,Z 177,A 90.5196,B 6.5845,C 0.1178,E1 6.5887,E2 361.8749} C_DIS
LIN {X -1.8503,Y 141.1833,Z 177,A 92.0574,B 6.5845,C 0.1205,E1 6.5845,E2 360.3611} C_DIS
LIN {X -4.6534,Y 141.1197,Z 177,A 93.2468,B 6.5845,C 0.1198,E1 6.5811,E2 359.1657} C_DIS
LIN {X -7.8774,Y 140.9767,Z 177,A 94.566,B 6.5845,C 0.1198,E1 6.5774,E2 357.8459} C_DIS
LIN {X -10.3689,Y 140.8132,Z 177,A 95.6307,B 6.5845,C 0.1193,E1 6.5745,E2 356.7751} C_DIS
LIN {X -13.6966,Y 140.5286,Z 177,A 96.9431,B 6.5845,C 0.1202,E1 6.5708,E2 355.4688} C_DIS
LIN {X -17.6919,Y 140.0831,Z 177,A 98.7046,B 6.5845,C 0.1189,E1 6.5659,E2 353.6916} C_DIS
LIN {X -22.4966,Y 139.3915,Z 177,A 101.0098,B 6.5845,C 0.1149,E1 6.5594,E2 351.3445} C_DIS
LIN {X -26.5057,Y 138.684,Z 177,A 102.7779,B 6.5846,C 0.1141,E1 6.5545,E2 349.5624} C_DIS
LIN {X -31.1634,Y 137.7125,Z 177,A 104.1167,B 6.5844,C 0.1237,E1 6.5511,E2 348.3007} C_DIS
LIN {X -37.8928,Y 136.0144,Z 177,A 107.1022,B 6.5844,C 0.1233,E1 6.543,E2 345.2955} C_DIS
LIN {X -42.393,Y 134.6809,Z 177,A 108.858,B 6.5844,C 0.1269,E1 6.5383,E2 343.5601} C_DIS
LIN {X -45.8333,Y 133.5487,Z 177,A 110.4865,B 6.5844,C 0.1261,E1 6.534,E2 341.9123} C_DIS
LIN {X -49.269,Y 132.3193,Z 177,A 112.0387,B 6.5844,C 0.1265,E1 6.5299,E2 340.352} C_DIS
LIN {X -52.9634,Y 130.8841,Z 177,A 113.6133,B 6.5844,C 0.1287,E1 6.5258,E2 338.7829} C_DIS
LIN {X -56.4178,Y 129.4331,Z 177,A 115.0615,B 6.5843,C 0.1314,E1 6.5221,E2 337.3449} C_DIS
LIN {X -59.7477,Y 127.9305,Z 177,A 116.5588,B 6.5843,C 0.1329,E1 6.5183,E2 335.8469} C_DIS
LIN {X -63.2612,Y 126.232,Z 177,A 118.1526,B 6.5843,C 0.1348,E1 6.5143,E2 334.2531} C_DIS
LIN {X -66.867,Y 124.3587,Z 177,A 119.9138,B 6.5843,C 0.1355,E1 6.5099,E2 332.4788} C_DIS
LIN {X -71.0202,Y 122.0349,Z 177,A 121.8733,B 6.5842,C 0.1378,E1 6.5052,E2 330.5171} C_DIS
LIN {X -74.9857,Y 119.6396,Z 177,A 123.7799,B 6.5842,C 0.1403,E1 6.5006,E2 328.6087} C_DIS
LIN {X -78.8284,Y 117.1432,Z 177,A 125.6776,B 6.5841,C 0.1427,E1 6.4962,E2 326.7076} C_DIS
LIN {X -85.3147,Y 112.5069,Z 177,A 128.6577,B 6.5839,C 0.1515,E1 6.4896,E2 323.7629} C_DIS
LIN {X -87.7272,Y 110.6358,Z 177,A 130.1137,B 6.5839,C 0.1509,E1 6.4863,E2 322.2803} C_DIS
LIN {X -90.9649,Y 107.9895,Z 177,A 132.3107,B 6.5839,C 0.1476,E1 6.4815,E2 320.0205} C_DIS
LIN {X -94.3596,Y 105.0362,Z 177,A 133.871,B 6.5838,C 0.1545,E1 6.4783,E2 318.496} C_DIS
LIN {X -98.4224,Y 101.2393,Z 177,A 136.0213,B 6.5836,C 0.1603,E1 6.474,E2 316.3614} C_DIS
LIN {X -101.562,Y 98.0891,Z 177,A 138.2882,B 6.5836,C 0.1582,E1 6.4694,E2 314.0366} C_DIS
LIN {X -104.6304,Y 94.8092,Z 177,A 139.6922,B 6.5835,C 0.1673,E1 6.4669,E2 312.6882} C_DIS
LIN {X -108.8686,Y 89.9108,Z 177,A 142.2816,B 6.5833,C 0.1735,E1 6.4622,E2 310.1063} C_DIS
LIN {X -110.6261,Y 87.7394,Z 177,A 143.9449,B 6.5834,C 0.1695,E1 6.4592,E2 308.3758} C_DIS
LIN {X -113.2755,Y 84.2908,Z 177,A 144.9441,B 6.5831,C 0.183,E1 6.4577,E2 307.4767} C_DIS
LIN {X -116.2306,Y 80.1676,Z 177,A 147.375,B 6.5831,C 0.1833,E1 6.4537,E2 305.0001} C_DIS
LIN {X -118.6086,Y 76.6055,Z 177,A 149.2301,B 6.583,C 0.186,E1 6.4508,E2 303.1315} C_DIS
LIN {X -120.9845,Y 72.7952,Z 177,A 151.0808,B 6.5829,C 0.1901,E1 6.4481,E2 301.2789} C_DIS
LIN {X -123.2153,Y 68.9518,Z 177,A 152.8555,B 6.5827,C 0.195,E1 6.4457,E2 299.5095} C_DIS
LIN {X -125.7539,Y 64.2004,Z 177,A 155.32,B 6.5827,C 0.1972,E1 6.4425,E2 297.011} C_DIS
LIN {X -127.1971,Y 61.2931,Z 177,A 156.4509,B 6.5825,C 0.2028,E1 6.4411,E2 295.9054} C_DIS
LIN {X -128.4004,Y 58.7316,Z 177,A 157.567,B 6.5824,C 0.2062,E1 6.4398,E2 294.7946} C_DIS
LIN {X -129.9936,Y 55.1179,Z 177,A 159.6031,B 6.5824,C 0.2053,E1 6.4375,E2 292.704} C_DIS
LIN {X -131.429,Y 51.5983,Z 177,A 160.6361,B 6.5821,C 0.2155,E1 6.4365,E2 291.7382} C_DIS
LIN {X -132.3509,Y 49.1845,Z 177,A 161.7899,B 6.5821,C 0.217,E1 6.4354,E2 290.5718} C_DIS
LIN {X -133.5455,Y 45.8426,Z 177,A 163.3078,B 6.5819,C 0.22,E1 6.4339,E2 289.0452} C_DIS
LIN {X -134.622,Y 42.5775,Z 177,A 164.8862,B 6.5819,C 0.2217,E1 6.4326,E2 287.4444} C_DIS
LIN {X -135.7818,Y 38.7247,Z 177,A 166.3642,B 6.5817,C 0.228,E1 6.4314,E2 285.9879} C_DIS
LIN {X -136.5464,Y 35.9314,Z 177,A 167.577,B 6.5816,C 0.2308,E1 6.4306,E2 284.7713} C_DIS
LIN {X -137.3133,Y 32.8769,Z 177,A 168.9178,B 6.5815,C 0.2336,E1 6.4297,E2 283.4235} C_DIS
LIN {X -138.1125,Y 29.3418,Z 177,A 171.0695,B 6.5816,C 0.2297,E1 6.4284,E2 281.1845} C_DIS
LIN {X -139.1141,Y 24.1573,Z 177,A 172.5529,B 6.5811,C 0.2436,E1 6.4277,E2 279.789} C_DIS
LIN {X -139.6515,Y 20.8302,Z 177,A 173.9979,B 6.581,C 0.2466,E1 6.427,E2 278.3352} C_DIS
LIN {X -140.105,Y 17.5239,Z 177,A 175.9678,B 6.5811,C 0.2431,E1 6.4263,E2 276.2863} C_DIS
LIN {X -140.6189,Y 12.756,Z 177,A 177.5787,B 6.5808,C 0.2527,E1 6.4259,E2 274.7208} C_DIS
LIN {X -140.9726,Y 7.9448,Z 177,A 179.3529,B 6.5805,C 0.2604,E1 6.4256,E2 272.9721} C_DIS
LIN {X -141.105,Y 5.0463,Z 177,A -179.4349,B 6.5803,C 0.2634,E1 6.4255,E2 271.7564} C_DIS
LIN {X -141.1879,Y 1.5662,Z 177,A -177.649,B 6.5803,C 0.263,E1 6.4255,E2 269.923} C_DIS
LIN {X -141.1846,Y -1.7577,Z 177,A -176.2788,B 6.5803,C 0.2666,E1 6.4255,E2 268.5511} C_DIS
LIN {X -141.1036,Y -5.0833,Z 177,A -175.3626,B 6.5798,C 0.2756,E1 6.4255,E2 267.6925} C_DIS
LIN {X -140.9677,Y -8.0258,Z 177,A -173.9701,B 6.5798,C 0.2767,E1 6.4257,E2 266.2754} C_DIS
LIN {X -140.743,Y -11.2963,Z 177,A -171.9859,B 6.58,C 0.2727,E1 6.4262,E2 264.2064} C_DIS
LIN {X -140.2412,Y -16.3821,Z 177,A -170.6381,B 6.5794,C 0.2873,E1 6.4266,E2 262.9555} C_DIS
LIN {X -139.8699,Y -19.3051,Z 177,A -168.9654,B 6.5794,C 0.285,E1 6.4272,E2 261.2212} C_DIS
LIN {X -139.368,Y -22.6438,Z 177,A -167.9691,B 6.5791,C 0.2933,E1 6.4276,E2 260.275} C_DIS
LIN {X -138.7546,Y -26.1366,Z 177,A -166.5093,B 6.5789,C 0.2971,E1 6.4284,E2 258.8135} C_DIS
LIN {X -138.188,Y -28.9921,Z 177,A -165.2097,B 6.5789,C 0.299,E1 6.4291,E2 257.4993} C_DIS
LIN {X -137.5157,Y -32.0249,Z 177,A -163.9187,B 6.5787,C 0.3021,E1 6.4299,E2 256.2052} C_DIS
LIN {X -136.8165,Y -34.8863,Z 177,A -162.6868,B 6.5786,C 0.305,E1 6.4307,E2 254.9692} C_DIS
LIN {X -135.9236,Y -38.2176,Z 177,A -161.2362,B 6.5784,C 0.3082,E1 6.4318,E2 253.5129} C_DIS
LIN {X -134.6689,Y -42.4306,Z 177,A -159.5111,B 6.5781,C 0.3137,E1 6.4332,E2 251.7967} C_DIS
LIN {X -133.7632,Y -45.2058,Z 177,A -158.2148,B 6.5781,C 0.3156,E1 6.4344,E2 250.4865} C_DIS
LIN {X -130.388,Y -54.1734,Z 177,A -154.4741,B 6.5775,C 0.3277,E1 6.4381,E2 246.7678} C_DIS
LIN {X -128.2548,Y -59.0466,Z 177,A -152.2799,B 6.5772,C 0.3329,E1 6.4406,E2 244.5703} C_DIS
LIN {X -127.226,Y -61.2326,Z 177,A -151.0423,B 6.5772,C 0.3322,E1 6.4421,E2 243.2994} C_DIS
LIN {X -125.4993,Y -64.7006,Z 177,A -149.4379,B 6.5771,C 0.3358,E1 6.4441,E2 241.6916} C_DIS
LIN {X -122.2197,Y -70.7011,Z 177,A -146.7621,B 6.5766,C 0.3439,E1 6.4477,E2 239.0304} C_DIS
LIN {X -120.6944,Y -73.2749,Z 177,A -145.2831,B 6.5766,C 0.3435,E1 6.4499,E2 237.517} C_DIS
LIN {X -118.1295,Y -77.3423,Z 177,A -143.528,B 6.5763,C 0.3506,E1 6.4525,E2 235.7887} C_DIS
LIN {X -116.3329,Y -80.0185,Z 177,A -141.9782,B 6.5763,C 0.3506,E1 6.455,E2 234.2074} C_DIS
LIN {X -113.7391,Y -83.6643,Z 177,A -140.1242,B 6.5761,C 0.3542,E1 6.458,E2 232.3491} C_DIS
LIN {X -110.9887,Y -87.28,Z 177,A -138.2265,B 6.5759,C 0.3576,E1 6.4613,E2 230.4449} C_DIS
LIN {X -108.2196,Y -90.6908,Z 177,A -136.425,B 6.5757,C 0.3611,E1 6.4645,E2 228.6415} C_DIS
LIN {X -105.1286,Y -94.2564,Z 177,A -134.5167,B 6.5755,C 0.3652,E1 6.468,E2 226.7347} C_DIS
LIN {X -102.2516,Y -97.3702,Z 177,A -132.7539,B 6.5753,C 0.3681,E1 6.4714,E2 224.9667} C_DIS
LIN {X -99.2903,Y -100.3883,Z 177,A -131.0103,B 6.5752,C 0.3711,E1 6.4748,E2 223.2199} C_DIS
LIN {X -96.131,Y -103.4173,Z 177,A -129.2096,B 6.575,C 0.3742,E1 6.4785,E2 221.4163} C_DIS
LIN {X -92.8051,Y -106.4119,Z 177,A -127.334,B 6.5749,C 0.3767,E1 6.4824,E2 219.5331} C_DIS
LIN {X -89.3237,Y -109.3506,Z 177,A -125.4855,B 6.5747,C 0.3799,E1 6.4864,E2 217.685} C_DIS
LIN {X -85.7478,Y -112.1767,Z 177,A -123.6051,B 6.5745,C 0.3826,E1 6.4905,E2 215.8008} C_DIS
LIN {X -81.9,Y -115.0163,Z 177,A -121.8185,B 6.5742,C 0.3878,E1 6.4945,E2 214.0349} C_DIS
LIN {X -79.3699,Y -116.7766,Z 177,A -120.4482,B 6.5742,C 0.3881,E1 6.4977,E2 212.6487} C_DIS
LIN {X -75.9044,Y -119.0583,Z 177,A -118.7298,B 6.5741,C 0.3901,E1 6.5017,E2 210.9258} C_DIS
LIN {X -72.2238,Y -121.3261,Z 177,A -116.8822,B 6.5741,C 0.3912,E1 6.5062,E2 209.0657} C_DIS
LIN {X -68.0676,Y -123.7062,Z 177,A -114.9147,B 6.5739,C 0.3934,E1 6.511,E2 207.0951} C_DIS
LIN {X -64.096,Y -125.807,Z 177,A -113.1759,B 6.5737,C 0.3968,E1 6.5153,E2 205.3674} C_DIS
LIN {X -60.5742,Y -127.5405,Z 177,A -111.5216,B 6.5737,C 0.3978,E1 6.5195,E2 203.7048} C_DIS
LIN {X -56.7171,Y -129.3037,Z 177,A -109.8848,B 6.5734,C 0.4008,E1 6.5236,E2 202.0791} C_DIS
LIN {X -53.777,Y -130.5536,Z 177,A -108.5399,B 6.5734,C 0.4014,E1 6.5271,E2 200.7276} C_DIS
LIN {X -50.7877,Y -131.7441,Z 177,A -107.0905,B 6.5734,C 0.4006,E1 6.5309,E2 199.2588} C_DIS
LIN {X -47.1561,Y -133.0889,Z 177,A -105.5464,B 6.5734,C 0.4023,E1 6.535,E2 197.7182} C_DIS
LIN {X -43.5275,Y -134.3185,Z 177,A -104.1194,B 6.5732,C 0.4054,E1 6.5387,E2 196.3079} C_DIS
LIN {X -40.537,Y -135.2523,Z 177,A -102.5052,B 6.5734,C 0.4013,E1 6.5431,E2 194.6474} C_DIS
LIN {X -37.3943,Y -136.1539,Z 177,A -101.3213,B 6.5732,C 0.4043,E1 6.5463,E2 193.4824} C_DIS
LIN {X -33.3386,Y -137.202,Z 177,A -99.6845,B 6.5732,C 0.4062,E1 6.5507,E2 191.8536} C_DIS
LIN {X -28.9478,Y -138.1972,Z 177,A -97.943,B 6.573,C 0.4083,E1 6.5554,E2 190.1232} C_DIS
LIN {X -25.4919,Y -138.8754,Z 177,A -96.3218,B 6.5731,C 0.4061,E1 6.5599,E2 188.4757} C_DIS
LIN {X -21.3747,Y -139.5672,Z 177,A -94.7817,B 6.5729,C 0.4089,E1 6.5641,E2 186.9557} C_DIS
LIN {X -17.1637,Y -140.1479,Z 177,A -93.0834,B 6.5729,C 0.4098,E1 6.5688,E2 185.2604} C_DIS
LIN {X -14.0988,Y -140.49,Z 177,A -91.8943,B 6.5729,C 0.411,E1 6.5721,E2 184.0792} C_DIS
LIN {X -11.2498,Y -140.7469,Z 177,A -90.6717,B 6.5729,C 0.4102,E1 6.5755,E2 182.8479} C_DIS
LIN {X -8.2055,Y -140.9566,Z 177,A -89.2578,B 6.573,C 0.4075,E1 6.5795,E2 181.4098} C_DIS
LIN {X -3.8136,Y -141.143,Z 177,A -87.5879,B 6.573,C 0.4092,E1 6.5842,E2 179.7545} C_DIS
LIN {X -0.2135,Y -141.1955,Z 177,A -86.1982,B 6.5729,C 0.4102,E1 6.588,E2 178.3737} C_DIS
LIN {X -0.2135,Y -141.1955,Z 177,A -86.1982,B 6.5729,C 0.4102,E1 6.588,E2 178.3737} C_DIS
Enddeposition()
LIN {X 1.0178,Y -142.0948,Z 177,A -85.9796,B 6.5723,C 0.4182,E1 6.5884,E2 178.2253} C_DIS
Startdeposition()
$VEL.CP = VEL_PRINT
LIN {X -1.7435,Y -142.0899,Z 177,A -87.384,B 6.572,C 0.4229,E1 6.5843,E2 179.6695} C_DIS
LIN {X -5.2371,Y -142.003,Z 177,A -88.7826,B 6.572,C 0.4227,E1 6.5804,E2 181.0674} C_DIS
LIN {X -8.7374,Y -141.8303,Z 177,A -90.1877,B 6.572,C 0.4226,E1 6.5765,E2 182.4719} C_DIS
LIN {X -12.1976,Y -141.5749,Z 177,A -91.5828,B 6.572,C 0.4224,E1 6.5726,E2 183.867} C_DIS
LIN {X -15.6626,Y -141.2341,Z 177,A -93.0022,B 6.572,C 0.4224,E1 6.5687,E2 185.2891} C_DIS
LIN {X -19.119,Y -140.8086,Z 177,A -94.3894,B 6.572,C 0.4218,E1 6.5648,E2 186.6746} C_DIS
LIN {X -22.5776,Y -140.2963,Z 177,A -95.832,B 6.572,C 0.4218,E1 6.5608,E2 188.1221} C_DIS
LIN {X -26.025,Y -139.6971,Z 177,A -97.2377,B 6.5721,C 0.4212,E1 6.557,E2 189.5275} C_DIS
LIN {X -29.718,Y -138.957,Z 177,A -98.6756,B 6.5722,C 0.4193,E1 6.5531,E2 190.955} C_DIS
LIN {X -32.8403,Y -138.2528,Z 177,A -100.0557,B 6.5722,C 0.4199,E1 6.5493,E2 192.3475} C_DIS
LIN {X -36.219,Y -137.4061,Z 177,A -101.4589,B 6.5722,C 0.4191,E1 6.5455,E2 193.7508} C_DIS
LIN {X -39.5531,Y -136.4837,Z 177,A -102.8775,B 6.5722,C 0.4185,E1 6.5417,E2 195.1729} C_DIS
LIN {X -42.9356,Y -135.4574,Z 177,A -104.3902,B 6.5722,C 0.4187,E1 6.5376,E2 196.6976} C_DIS
LIN {X -47.2605,Y -134.0115,Z 177,A -106.2291,B 6.5724,C 0.4172,E1 6.5327,E2 198.5369} C_DIS
LIN {X -51.1494,Y -132.5742,Z 177,A -107.8272,B 6.5725,C 0.4146,E1 6.5286,E2 200.1253} C_DIS
LIN {X -54.3764,Y -131.2838,Z 177,A -109.2447,B 6.5725,C 0.4135,E1 6.5249,E2 201.5452} C_DIS
LIN {X -57.597,Y -129.9032,Z 177,A -110.6607,B 6.5727,C 0.4121,E1 6.5213,E2 202.9618} C_DIS
LIN {X -61.259,Y -128.2161,Z 177,A -112.3558,B 6.5727,C 0.4112,E1 6.517,E2 204.6662} C_DIS
LIN {X -64.6597,Y -126.5354,Z 177,A -113.8556,B 6.5729,C 0.409,E1 6.5132,E2 206.162} C_DIS
LIN {X -67.7555,Y -124.9076,Z 177,A -115.2714,B 6.5729,C 0.4073,E1 6.5097,E2 207.5787} C_DIS
LIN {X -70.8042,Y -123.2054,Z 177,A -116.7016,B 6.5731,C 0.4058,E1 6.5063,E2 209.0119} C_DIS
LIN {X -73.7987,Y -121.435,Z 177,A -118.1379,B 6.5731,C 0.4043,E1 6.5028,E2 210.4527} C_DIS
LIN {X -77.4942,Y -119.1104,Z 177,A -119.9367,B 6.5733,C 0.4023,E1 6.4986,E2 212.2565} C_DIS
LIN {X -81.1071,Y -116.6802,Z 177,A -121.6674,B 6.5735,C 0.3993,E1 6.4946,E2 213.9837} C_DIS
LIN {X -84.0326,Y -114.5912,Z 177,A -123.1131,B 6.5736,C 0.3969,E1 6.4913,E2 215.4288} C_DIS
LIN {X -87.2474,Y -112.1631,Z 177,A -124.817,B 6.5737,C 0.3953,E1 6.4875,E2 217.1431} C_DIS
LIN {X -90.1505,Y -109.8434,Z 177,A -126.3074,B 6.5739,C 0.3926,E1 6.4843,E2 218.6322} C_DIS
LIN {X -92.8162,Y -107.6,Z 177,A -127.8623,B 6.5739,C 0.3921,E1 6.4809,E2 220.2067} C_DIS
LIN {X -96.0887,Y -104.688,Z 177,A -129.5139,B 6.5742,C 0.3874,E1 6.4775,E2 221.8427} C_DIS
LIN {X -98.6208,Y -102.3066,Z 177,A -130.9353,B 6.5743,C 0.385,E1 6.4747,E2 223.2664} C_DIS
LIN {X -101.0981,Y -99.8596,Z 177,A -132.3745,B 6.5745,C 0.3827,E1 6.4718,E2 224.71} C_DIS
LIN {X -103.5143,Y -97.3521,Z 177,A -133.797,B 6.5746,C 0.3801,E1 6.4691,E2 226.1345} C_DIS
LIN {X -105.8725,Y -94.7819,Z 177,A -135.2201,B 6.5748,C 0.3774,E1 6.4664,E2 227.5594} C_DIS
LIN {X -108.6482,Y -91.5876,Z 177,A -136.985,B 6.5749,C 0.3746,E1 6.4632,E2 229.3315} C_DIS
LIN {X -110.9499,Y -88.7855,Z 177,A -138.4368,B 6.5751,C 0.3713,E1 6.4606,E2 230.7814} C_DIS
LIN {X -113.093,Y -86.039,Z 177,A -139.8791,B 6.5753,C 0.3687,E1 6.4581,E2 232.2282} C_DIS
LIN {X -115.1718,Y -83.2352,Z 177,A -141.3066,B 6.5754,C 0.3657,E1 6.4558,E2 233.6577} C_DIS
LIN {X -117.1773,Y -80.3871,Z 177,A -142.7333,B 6.5756,C 0.3628,E1 6.4535,E2 235.0868} C_DIS
LIN {X -119.124,Y -77.4731,Z 177,A -144.1685,B 6.5757,C 0.3598,E1 6.4513,E2 236.5244} C_DIS
LIN {X -120.9807,Y -74.5409,Z 177,A -145.5916,B 6.5759,C 0.3567,E1 6.4492,E2 237.95} C_DIS
LIN {X -122.7631,Y -71.5682,Z 177,A -147.0256,B 6.5761,C 0.3538,E1 6.4471,E2 239.3881} C_DIS
LIN {X -124.4785,Y -68.5407,Z 177,A -148.4614,B 6.5762,C 0.3508,E1 6.4452,E2 240.8275} C_DIS
LIN {X -126.1355,Y -65.4398,Z 177,A -149.9072,B 6.5764,C 0.3476,E1 6.4433,E2 242.2762} C_DIS
LIN {X -127.7017,Y -62.327,Z 177,A -151.3379,B 6.5766,C 0.3443,E1 6.4415,E2 243.7095} C_DIS
LIN {X -129.5213,Y -58.4508,Z 177,A -153.1168,B 6.5768,C 0.3405,E1 6.4394,E2 245.4943} C_DIS
LIN {X -130.8321,Y -55.4579,Z 177,A -154.3962,B 6.577,C 0.3367,E1 6.438,E2 246.768} C_DIS
LIN {X -131.9281,Y -52.7936,Z 177,A -155.6242,B 6.577,C 0.3344,E1 6.4367,E2 248.004} C_DIS
LIN {X -133.1804,Y -49.5493,Z 177,A -157.0625,B 6.5772,C 0.3311,E1 6.4353,E2 249.4462} C_DIS
LIN {X -134.3727,Y -46.2188,Z 177,A -158.512,B 6.5774,C 0.3276,E1 6.4339,E2 250.8978} C_DIS
LIN {X -135.4648,Y -42.9126,Z 177,A -159.9465,B 6.5776,C 0.3242,E1 6.4327,E2 252.3354} C_DIS
LIN {X -136.4791,Y -39.5688,Z 177,A -161.3825,B 6.5778,C 0.3206,E1 6.4316,E2 253.774} C_DIS
LIN {X -137.4876,Y -35.9135,Z 177,A -162.9332,B 6.5779,C 0.3167,E1 6.4304,E2 255.3267} C_DIS
LIN {X -138.2588,Y -32.8157,Z 177,A -164.2574,B 6.5781,C 0.3136,E1 6.4296,E2 256.6548} C_DIS
LIN {X -139.0195,Y -29.4282,Z 177,A -165.6867,B 6.5783,C 0.31,E1 6.4287,E2 258.0869} C_DIS
LIN {X -139.81,Y -25.4056,Z 177,A -167.2058,B 6.5786,C 0.3038,E1 6.4279,E2 259.5873} C_DIS
LIN {X -140.2896,Y -22.6182,Z 177,A -168.5358,B 6.5786,C 0.3029,E1 6.4273,E2 260.9413} C_DIS
LIN {X -140.7935,Y -19.2336,Z 177,A -169.969,B 6.5787,C 0.2996,E1 6.4267,E2 262.3804} C_DIS
LIN {X -141.2228,Y -15.7673,Z 177,A -171.4098,B 6.5789,C 0.296,E1 6.4262,E2 263.8244} C_DIS
LIN {X -141.5812,Y -12.1231,Z 177,A -172.9884,B 6.579,C 0.293,E1 6.4258,E2 265.4151} C_DIS
LIN {X -141.8311,Y -8.7247,Z 177,A -174.3105,B 6.5792,C 0.2885,E1 6.4256,E2 266.7293} C_DIS
LIN {X -142.0027,Y -5.2456,Z 177,A -175.7383,B 6.5794,C 0.2847,E1 6.4254,E2 268.159} C_DIS
LIN {X -142.0896,Y -1.7665,Z 177,A -177.1143,B 6.5796,C 0.2804,E1 6.4254,E2 269.5304} C_DIS
LIN {X -142.0898,Y 1.7501,Z 177,A -178.7446,B 6.5796,C 0.2788,E1 6.4254,E2 271.187} C_DIS
LIN {X -142.0032,Y 5.2322,Z 177,A 179.9214,B 6.5799,C 0.274,E1 6.4254,E2 272.5108} C_DIS
LIN {X -141.8327,Y 8.6985,Z 177,A 178.4976,B 6.58,C 0.2702,E1 6.4257,E2 273.9365} C_DIS
LIN {X -141.5788,Y 12.1513,Z 177,A 177.0738,B 6.5802,C 0.2666,E1 6.426,E2 275.3628} C_DIS
LIN {X -141.1764,Y 16.181,Z 177,A 175.3998,B 6.5803,C 0.2624,E1 6.4265,E2 277.0408} C_DIS
LIN {X -140.8093,Y 19.113,Z 177,A 174.1939,B 6.5805,C 0.2592,E1 6.427,E2 278.2475} C_DIS
LIN {X -140.2997,Y 22.5564,Z 177,A 172.7396,B 6.5805,C 0.2558,E1 6.4276,E2 279.7071} C_DIS
LIN {X -139.7067,Y 25.9748,Z 177,A 171.3054,B 6.5807,C 0.2523,E1 6.4283,E2 281.1446} C_DIS
LIN {X -139.0158,Y 29.4455,Z 177,A 169.8543,B 6.5809,C 0.2485,E1 6.4291,E2 282.5975} C_DIS
LIN {X -138.1906,Y 33.0985,Z 177,A 168.3726,B 6.581,C 0.244,E1 6.43,E2 284.0742} C_DIS
LIN {X -137.4001,Y 36.2419,Z 177,A 166.9787,B 6.5811,C 0.2414,E1 6.431,E2 285.4781} C_DIS
LIN {X -136.474,Y 39.5861,Z 177,A 165.5435,B 6.5813,C 0.2379,E1 6.4321,E2 286.9167} C_DIS
LIN {X -135.3459,Y 43.2848,Z 177,A 164.0365,B 6.5814,C 0.233,E1 6.4333,E2 288.4156} C_DIS
LIN {X -134.3631,Y 46.2463,Z 177,A 162.6733,B 6.5815,C 0.2308,E1 6.4346,E2 289.7911} C_DIS
LIN {X -133.1909,Y 49.5213,Z 177,A 161.2385,B 6.5816,C 0.2274,E1 6.4359,E2 291.2288} C_DIS
LIN {X -131.6498,Y 53.484,Z 177,A 159.6264,B 6.5818,C 0.2216,E1 6.4376,E2 292.8262} C_DIS
LIN {X -130.5801,Y 56.0449,Z 177,A 158.3656,B 6.5818,C 0.2204,E1 6.439,E2 294.1042} C_DIS
LIN {X -129.2024,Y 59.153,Z 177,A 156.95,B 6.582,C 0.2173,E1 6.4406,E2 295.5243} C_DIS
LIN {X -127.7176,Y 62.2948,Z 177,A 155.5228,B 6.582,C 0.214,E1 6.4423,E2 296.9535} C_DIS
LIN {X -126.1562,Y 65.4003,Z 177,A 153.981,B 6.5821,C 0.2121,E1 6.4443,E2 298.5119} C_DIS
LIN {X -124.0644,Y 69.2877,Z 177,A 152.2746,B 6.5823,C 0.2067,E1 6.4466,E2 300.2074} C_DIS
LIN {X -122.3289,Y 72.3077,Z 177,A 150.8329,B 6.5823,C 0.2037,E1 6.4486,E2 301.6525} C_DIS
LIN {X -120.5196,Y 75.2842,Z 177,A 149.4034,B 6.5825,C 0.2005,E1 6.4507,E2 303.0839} C_DIS
LIN {X -118.5609,Y 78.3324,Z 177,A 147.7765,B 6.5825,C 0.199,E1 6.4532,E2 304.7306} C_DIS
LIN {X -116.1749,Y 81.8291,Z 177,A 146.1821,B 6.5827,C 0.1936,E1 6.4557,E2 306.3091} C_DIS
LIN {X -113.9561,Y 84.8918,Z 177,A 144.5253,B 6.5827,C 0.1917,E1 6.4585,E2 307.9814} C_DIS
LIN {X -111.1162,Y 88.5766,Z 177,A 142.6738,B 6.5829,C 0.1872,E1 6.4617,E2 309.828} C_DIS
LIN {X -108.7514,Y 91.4645,Z 177,A 141.1849,B 6.5829,C 0.1836,E1 6.4643,E2 311.3135} C_DIS
LIN {X -106.4965,Y 94.0803,Z 177,A 139.772,B 6.5831,C 0.1809,E1 6.4669,E2 312.7278} C_DIS
LIN {X -104.1546,Y 96.6668,Z 177,A 138.3259,B 6.5831,C 0.1784,E1 6.4696,E2 314.1776} C_DIS
LIN {X -101.7017,Y 99.2447,Z 177,A 136.8904,B 6.5832,C 0.1754,E1 6.4724,E2 315.6119} C_DIS
LIN {X -99.2468,Y 101.6996,Z 177,A 135.4528,B 6.5832,C 0.1731,E1 6.4753,E2 317.0531} C_DIS
LIN {X -96.7363,Y 104.0899,Z 177,A 134.0366,B 6.5833,C 0.1706,E1 6.4782,E2 318.4704} C_DIS
LIN {X -94.1582,Y 106.4277,Z 177,A 132.6045,B 6.5833,C 0.1682,E1 6.4812,E2 319.9049} C_DIS
LIN {X -90.9224,Y 109.2056,Z 177,A 130.845,B 6.5835,C 0.1656,E1 6.4849,E2 321.6681} C_DIS
LIN {X -88.1302,Y 111.4714,Z 177,A 129.3939,B 6.5835,C 0.163,E1 6.4881,E2 323.118} C_DIS
LIN {X -85.3822,Y 113.5894,Z 177,A 127.9775,B 6.5835,C 0.1608,E1 6.4912,E2 324.5355} C_DIS
LIN {X -82.5751,Y 115.6459,Z 177,A 126.4238,B 6.5835,C 0.1604,E1 6.4948,E2 326.1071} C_DIS
LIN {X -78.9379,Y 118.1585,Z 177,A 124.7553,B 6.5837,C 0.156,E1 6.4986,E2 327.7597} C_DIS
LIN {X -76.0176,Y 120.0582,Z 177,A 123.3355,B 6.5837,C 0.1541,E1 6.5019,E2 329.1803} C_DIS
LIN {X -73.0517,Y 121.886,Z 177,A 121.9177,B 6.5837,C 0.1522,E1 6.5053,E2 330.5986} C_DIS
LIN {X -69.7611,Y 123.7983,Z 177,A 120.268,B 6.5837,C 0.1515,E1 6.5093,E2 332.2617} C_DIS
LIN {X -66.214,Y 125.7289,Z 177,A 118.719,B 6.5839,C 0.1482,E1 6.5131,E2 333.7993} C_DIS
LIN {X -63.0955,Y 127.3227,Z 177,A 117.2927,B 6.5839,C 0.1466,E1 6.5167,E2 335.2263} C_DIS
LIN {X -59.9562,Y 128.8309,Z 177,A 115.8736,B 6.5839,C 0.1451,E1 6.5203,E2 336.6463} C_DIS
LIN {X -57.5766,Y 129.9123,Z 177,A 114.805,B 6.5839,C 0.1441,E1 6.523,E2 337.716} C_DIS
LIN {X -54.3806,Y 131.282,Z 177,A 113.3934,B 6.5839,C 0.1427,E1 6.5266,E2 339.1278} C_DIS
LIN {X -51.1629,Y 132.569,Z 177,A 111.9801,B 6.584,C 0.1414,E1 6.5303,E2 340.5421} C_DIS
LIN {X -47.8744,Y 133.7917,Z 177,A 110.5157,B 6.584,C 0.1407,E1 6.5342,E2 342.0118} C_DIS
LIN {X -44.5695,Y 134.9287,Z 177,A 109.1408,B 6.584,C 0.139,E1 6.5378,E2 343.3814} C_DIS
LIN {X -41.238,Y 135.984,Z 177,A 107.7236,B 6.584,C 0.1379,E1 6.5416,E2 344.7987} C_DIS
LIN {X -37.8558,Y 136.9643,Z 177,A 106.2974,B 6.5841,C 0.1369,E1 6.5454,E2 346.2248} C_DIS
LIN {X -34.4993,Y 137.8482,Z 177,A 104.8918,B 6.5841,C 0.136,E1 6.5492,E2 347.6303} C_DIS
LIN {X -31.1486,Y 138.6439,Z 177,A 103.4975,B 6.5841,C 0.1352,E1 6.553,E2 349.0245} C_DIS
LIN {X -27.7625,Y 139.3618,Z 177,A 102.0975,B 6.5841,C 0.1345,E1 6.5568,E2 350.4242} C_DIS
LIN {X -24.3488,Y 139.9991,Z 177,A 100.6943,B 6.5841,C 0.1339,E1 6.5607,E2 351.827} C_DIS
LIN {X -20.8352,Y 140.5653,Z 177,A 99.2321,B 6.5841,C 0.1337,E1 6.5647,E2 353.2919} C_DIS
LIN {X -17.3863,Y 141.0326,Z 177,A 97.8271,B 6.5841,C 0.1332,E1 6.5686,E2 354.6963} C_DIS
LIN {X -13.928,Y 141.4154,Z 177,A 96.4276,B 6.5842,C 0.1327,E1 6.5725,E2 356.0946} C_DIS
LIN {X -10.0996,Y 141.74,Z 177,A 94.9361,B 6.5842,C 0.1316,E1 6.5766,E2 357.578} C_DIS
LIN {X -6.2497,Y 141.9635,Z 177,A 93.3794,B 6.5842,C 0.1314,E1 6.581,E2 359.1342} C_DIS
LIN {X -3.4731,Y 142.0576,Z 177,A 92.2201,B 6.5842,C 0.1319,E1 6.5842,E2 360.2979} C_DIS
LIN {X -0.0055,Y 142.1014,Z 177,A 90.7817,B 6.5842,C 0.1325,E1 6.5883,E2 361.7408} C_DIS
LIN {X 3.4771,Y 142.0575,Z 177,A 89.3844,B 6.5842,C 0.1325,E1 6.5922,E2 363.1366} C_DIS
LIN {X 7.7309,Y 141.89,Z 177,A 87.7527,B 6.5842,C 0.1315,E1 6.5967,E2 364.7568} C_DIS
LIN {X 10.4686,Y 141.7131,Z 177,A 86.5869,B 6.5842,C 0.1326,E1 6.5999,E2 365.9298} C_DIS
LIN {X 14.0452,Y 141.4041,Z 177,A 85.1564,B 6.5842,C 0.1327,E1 6.6039,E2 367.3576} C_DIS
LIN {X 17.3852,Y 141.0327,Z 177,A 83.7963,B 6.5842,C 0.1333,E1 6.6077,E2 368.7179} C_DIS
LIN {X 20.8583,Y 140.5619,Z 177,A 82.3806,B 6.5842,C 0.1339,E1 6.6116,E2 370.1334} C_DIS
LIN {X 24.3056,Y 140.0068,Z 177,A 80.869,B 6.5842,C 0.1362,E1 6.6158,E2 371.6578} C_DIS
LIN {X 27.7254,Y 139.3693,Z 177,A 79.571,B 6.5842,C 0.1354,E1 6.6193,E2 372.9421} C_DIS
LIN {X 31.3301,Y 138.6025,Z 177,A 78.1505,B 6.5842,C 0.1353,E1 6.6232,E2 374.3538} C_DIS
LIN {X 34.5212,Y 137.8426,Z 177,A 76.6391,B 6.5841,C 0.1391,E1 6.6273,E2 375.8889} C_DIS
LIN {X 38.2524,Y 136.8534,Z 177,A 75.314,B 6.5841,C 0.1367,E1 6.6308,E2 377.1842} C_DIS
LIN {X 41.2686,Y 135.9746,Z 177,A 73.9757,B 6.5841,C 0.1389,E1 6.6344,E2 378.5314} C_DIS
LIN {X 44.5894,Y 134.9221,Z 177,A 72.5812,B 6.5841,C 0.14,E1 6.6381,E2 379.9244} C_DIS
LIN {X 48.5339,Y 133.5539,Z 177,A 71.0306,B 6.5841,C 0.1395,E1 6.6422,E2 381.4578} C_DIS
LIN {X 51.1495,Y 132.5742,Z 177,A 69.7934,B 6.584,C 0.1424,E1 6.6455,E2 382.709} C_DIS
LIN {X 54.386,Y 131.2798,Z 177,A 68.4024,B 6.584,C 0.1437,E1 6.6491,E2 384.098} C_DIS
LIN {X 57.5892,Y 129.9067,Z 177,A 67.0126,B 6.584,C 0.1451,E1 6.6526,E2 385.4858} C_DIS
LIN {X 60.7528,Y 128.458,Z 177,A 65.6225,B 6.584,C 0.1466,E1 6.6561,E2 386.8741} C_DIS
LIN {X 63.8783,Y 126.9331,Z 177,A 64.2491,B 6.5839,C 0.1479,E1 6.6595,E2 388.2438} C_DIS
LIN {X 66.9221,Y 125.3562,Z 177,A 62.8461,B 6.5839,C 0.1501,E1 6.663,E2 389.6494} C_DIS
LIN {X 70.0397,Y 123.6416,Z 177,A 61.3238,B 6.5837,C 0.1536,E1 6.6668,E2 391.1829} C_DIS
LIN {X 73.8055,Y 121.4309,Z 177,A 59.6952,B 6.5837,C 0.154,E1 6.6706,E2 392.7947} C_DIS
LIN {X 76.7734,Y 119.5763,Z 177,A 58.3053,B 6.5837,C 0.1558,E1 6.6739,E2 394.182} C_DIS
LIN {X 79.6631,Y 117.6708,Z 177,A 56.8907,B 6.5837,C 0.1584,E1 6.6772,E2 395.5991} C_DIS
LIN {X 83.2445,Y 115.1651,Z 177,A 55.0952,B 6.5836,C 0.1619,E1 6.6813,E2 397.3991} C_DIS
LIN {X 86.7403,Y 112.5562,Z 177,A 53.4539,B 6.5836,C 0.1629,E1 6.6849,E2 399.0256} C_DIS
LIN {X 89.4743,Y 110.3951,Z 177,A 52.0592,B 6.5835,C 0.1653,E1 6.688,E2 400.4191} C_DIS
LIN {X 92.1634,Y 108.1598,Z 177,A 50.8179,B 6.5835,C 0.165,E1 6.6906,E2 401.639} C_DIS
LIN {X 94.7563,Y 105.8955,Z 177,A 49.3111,B 6.5834,C 0.1697,E1 6.6938,E2 403.1613} C_DIS
LIN {X 97.3039,Y 103.5599,Z 177,A 47.9416,B 6.5833,C 0.172,E1 6.6966,E2 404.5281} C_DIS
LIN {X 100.2042,Y 100.7558,Z 177,A 46.2729,B 6.5832,C 0.176,E1 6.6999,E2 406.2026} C_DIS
LIN {X 102.9184,Y 97.982,Z 177,A 44.788,B 6.5832,C 0.1778,E1 6.7028,E2 407.6777} C_DIS
LIN {X 105.289,Y 95.4298,Z 177,A 43.3824,B 6.5831,C 0.1808,E1 6.7054,E2 409.0838} C_DIS
LIN {X 108.1502,Y 92.1747,Z 177,A 41.6994,B 6.583,C 0.1835,E1 6.7085,E2 410.7591} C_DIS
LIN {X 110.3608,Y 89.5168,Z 177,A 40.3243,B 6.583,C 0.1862,E1 6.7109,E2 412.1322} C_DIS
LIN {X 112.5074,Y 86.8032,Z 177,A 38.9331,B 6.5828,C 0.1893,E1 6.7133,E2 413.5234} C_DIS
LIN {X 114.658,Y 83.9417,Z 177,A 37.4364,B 6.5828,C 0.1935,E1 6.7158,E2 415.0276} C_DIS
LIN {X 117.1832,Y 80.3785,Z 177,A 35.8022,B 6.5826,C 0.1955,E1 6.7184,E2 416.646} C_DIS
LIN {X 119.1165,Y 77.4848,Z 177,A 34.4271,B 6.5826,C 0.1983,E1 6.7205,E2 418.0182} C_DIS
LIN {X 120.9785,Y 74.5445,Z 177,A 33.0516,B 6.5825,C 0.2012,E1 6.7225,E2 419.3907} C_DIS
LIN {X 122.7655,Y 71.5641,Z 177,A 31.6686,B 6.5824,C 0.2043,E1 6.7245,E2 420.772} C_DIS
LIN {X 124.4953,Y 68.5103,Z 177,A 30.2781,B 6.5823,C 0.2074,E1 6.7264,E2 422.16} C_DIS
LIN {X 126.1347,Y 65.4412,Z 177,A 28.8996,B 6.5822,C 0.2105,E1 6.7282,E2 423.536} C_DIS
LIN {X 127.9767,Y 61.7601,Z 177,A 27.2168,B 6.582,C 0.2152,E1 6.7303,E2 425.2227} C_DIS
LIN {X 129.5528,Y 58.3804,Z 177,A 25.9694,B 6.582,C 0.2146,E1 6.7317,E2 426.4376} C_DIS
LIN {X 130.8509,Y 55.4129,Z 177,A 24.581,B 6.5819,C 0.2195,E1 6.7332,E2 427.8375} C_DIS
LIN {X 131.9342,Y 52.7785,Z 177,A 23.3939,B 6.5818,C 0.2232,E1 6.7345,E2 429.0302} C_DIS
LIN {X 133.2023,Y 49.4909,Z 177,A 22.0062,B 6.5817,C 0.2264,E1 6.7359,E2 430.4146} C_DIS
LIN {X 134.3716,Y 46.2219,Z 177,A 20.6344,B 6.5815,C 0.2297,E1 6.7371,E2 431.7835} C_DIS
LIN {X 135.4644,Y 42.9137,Z 177,A 19.2579,B 6.5815,C 0.233,E1 6.7383,E2 433.1573} C_DIS
LIN {X 136.6447,Y 38.9986,Z 177,A 17.6838,B 6.5813,C 0.2361,E1 6.7396,E2 434.7228} C_DIS
LIN {X 137.4141,Y 36.1891,Z 177,A 16.4956,B 6.5812,C 0.2396,E1 6.7404,E2 435.9135} C_DIS
LIN {X 138.2619,Y 32.8025,Z 177,A 15.1209,B 6.5811,C 0.2429,E1 6.7413,E2 437.2848} C_DIS
LIN {X 139.0211,Y 29.4207,Z 177,A 13.7542,B 6.5809,C 0.2463,E1 6.7421,E2 438.6485} C_DIS
LIN {X 139.7,Y 26.0097,Z 177,A 12.3354,B 6.5808,C 0.2505,E1 6.7429,E2 440.0704} C_DIS
LIN {X 140.2976,Y 22.5696,Z 177,A 10.9879,B 6.5807,C 0.2534,E1 6.7435,E2 441.4112} C_DIS
LIN {X 140.8073,Y 19.1286,Z 177,A 9.6039,B 6.5805,C 0.2571,E1 6.744,E2 442.7937} C_DIS
LIN {X 141.2365,Y 15.6402,Z 177,A 8.2293,B 6.5805,C 0.2603,E1 6.7445,E2 444.1638} C_DIS
LIN {X 141.5757,Y 12.1877,Z 177,A 6.7559,B 6.5802,C 0.2656,E1 6.7449,E2 445.6481} C_DIS
LIN {X 141.9278,Y 6.9786,Z 177,A 4.8141,B 6.5801,C 0.2687,E1 6.7452,E2 447.5701} C_DIS
LIN {X 142.0579,Y 3.4638,Z 177,A 3.3447,B 6.5799,C 0.2737,E1 6.7453,E2 449.0474} C_DIS
LIN {X 142.1032,Y 0,Z 177,A 1.8864,B 6.5797,C 0.2788,E1 6.7453,E2 450.5151} C_DIS
LIN {X 142.036,Y -4.2517,Z 177,A 0.5058,B 6.5797,C 0.2777,E1 6.7453,E2 451.853} C_DIS
LIN {X 141.9278,Y -6.9796,Z 177,A -0.7034,B 6.5795,C 0.2828,E1 6.7451,E2 453.0774} C_DIS
LIN {X 141.7124,Y -10.4793,Z 177,A -2.0787,B 6.5793,C 0.2861,E1 6.7448,E2 454.4489} C_DIS
LIN {X 141.4147,Y -13.9345,Z 177,A -3.4434,B 6.5792,C 0.2895,E1 6.7445,E2 455.8104} C_DIS
LIN {X 140.9498,Y -18.0411,Z 177,A -4.9287,B 6.5792,C 0.291,E1 6.744,E2 457.2732} C_DIS
LIN {X 140.564,Y -20.8437,Z 177,A -6.1913,B 6.5789,C 0.2965,E1 6.7435,E2 458.553} C_DIS
LIN {X 140.009,Y -24.2936,Z 177,A -7.588,B 6.5787,C 0.3002,E1 6.7429,E2 459.9493} C_DIS
LIN {X 139.3105,Y -28.0145,Z 177,A -9.0003,B 6.5787,C 0.3025,E1 6.7421,E2 461.3479} C_DIS
LIN {X 138.648,Y -31.1306,Z 177,A -10.3315,B 6.5784,C 0.3069,E1 6.7413,E2 462.6864} C_DIS
LIN {X 137.8435,Y -34.5178,Z 177,A -11.7045,B 6.5782,C 0.3103,E1 6.7404,E2 464.0565} C_DIS
LIN {X 136.9398,Y -37.9435,Z 177,A -13.0835,B 6.5782,C 0.3134,E1 6.7394,E2 465.4303} C_DIS
LIN {X 135.9892,Y -41.2211,Z 177,A -14.4611,B 6.5779,C 0.3172,E1 6.7383,E2 466.8094} C_DIS
LIN {X 134.9207,Y -44.5935,Z 177,A -15.8497,B 6.5778,C 0.3205,E1 6.7372,E2 468.1943} C_DIS
LIN {X 133.7864,Y -47.889,Z 177,A -17.2244,B 6.5776,C 0.3237,E1 6.7359,E2 469.5663} C_DIS
LIN {X 132.5689,Y -51.1631,Z 177,A -18.5976,B 6.5774,C 0.3269,E1 6.7345,E2 470.9361} C_DIS
LIN {X 131.2809,Y -54.3833,Z 177,A -19.9767,B 6.5773,C 0.3303,E1 6.7331,E2 472.314} C_DIS
LIN {X 129.9073,Y -57.5878,Z 177,A -21.3442,B 6.5771,C 0.3334,E1 6.7316,E2 473.6778} C_DIS
LIN {X 128.4581,Y -60.7526,Z 177,A -22.7201,B 6.577,C 0.3366,E1 6.7299,E2 475.0513} C_DIS
LIN {X 126.9313,Y -63.882,Z 177,A -24.0932,B 6.5768,C 0.3397,E1 6.7282,E2 476.4216} C_DIS
LIN {X 125.1188,Y -67.3641,Z 177,A -25.7225,B 6.5766,C 0.3446,E1 6.7261,E2 478.0586} C_DIS
LIN {X 123.2051,Y -70.8048,Z 177,A -27.2159,B 6.5764,C 0.3469,E1 6.7241,E2 479.541} C_DIS
LIN {X 121.4198,Y -73.8239,Z 177,A -28.6032,B 6.5763,C 0.35,E1 6.7221,E2 480.926} C_DIS
LIN {X 119.5799,Y -76.7678,Z 177,A -29.9743,B 6.5761,C 0.3529,E1 6.72,E2 482.2947} C_DIS
LIN {X 117.5489,Y -79.8431,Z 177,A -31.5471,B 6.5758,C 0.3581,E1 6.7176,E2 483.8805} C_DIS
LIN {X 115.1838,Y -83.2187,Z 177,A -33.059,B 6.5758,C 0.3594,E1 6.7152,E2 485.3739} C_DIS
LIN {X 113.1098,Y -86.0171,Z 177,A -34.4388,B 6.5756,C 0.3623,E1 6.7128,E2 486.7518} C_DIS
LIN {X 110.9422,Y -88.7951,Z 177,A -35.8451,B 6.5754,C 0.3653,E1 6.7104,E2 488.1575} C_DIS
LIN {X 108.7301,Y -91.4899,Z 177,A -37.2227,B 6.5753,C 0.368,E1 6.708,E2 489.5327} C_DIS
LIN {X 106.4609,Y -94.1206,Z 177,A -38.5962,B 6.5751,C 0.3706,E1 6.7054,E2 490.9037} C_DIS
LIN {X 104.119,Y -96.7051,Z 177,A -40.0369,B 6.5749,C 0.3743,E1 6.7027,E2 492.3504} C_DIS
LIN {X 101.0904,Y -99.8674,Z 177,A -41.7159,B 6.5749,C 0.3765,E1 6.6995,E2 494.0195} C_DIS
LIN {X 98.5549,Y -102.3703,Z 177,A -43.2774,B 6.5745,C 0.3817,E1 6.6963,E2 495.599} C_DIS
LIN {X 95.4334,Y -105.2857,Z 177,A -44.8267,B 6.5745,C 0.3821,E1 6.6932,E2 497.1268} C_DIS
LIN {X 92.6928,Y -107.7063,Z 177,A -46.4006,B 6.5742,C 0.3867,E1 6.6898,E2 498.7152} C_DIS
LIN {X 89.4686,Y -110.3996,Z 177,A -47.9404,B 6.5742,C 0.3873,E1 6.6865,E2 500.2359} C_DIS
LIN {X 86.7424,Y -112.5545,Z 177,A -49.3369,B 6.574,C 0.3898,E1 6.6835,E2 501.633} C_DIS
Enddeposition()
END
